(* IEC 61131-3 sources: std_i2980_v2.06_cp053/Source/IMM/ieccontrol/OperationMode1 (part 2) *)

(* ---- ABOperationMode.pu ---- *)
IMPORT_OVER_LISTFILE
 GET_ALARM_NAME
, SET_ALARM
, SET_EVENT
, tnOperationMode
, tsLockOperationModeAuto
, tsTraceLevel
, tnDataState
, ALARM_EVENT
, ABOpModeControl
, tevPanelButtonRegisterData
, tevPanelButtonRegister
, FBDebugTrace
, tsDeviceId
, ALARM_EVENT_DATA

END_IMPORT

ALGORITHM_BLOCK ABOperationMode #DUMMY_EDIT_BLOCK

SYSTEM_VAR
 di_ButtonSetup : BOOL;
 di_ButtonManual : BOOL;
 di_ButtonHalfAuto : BOOL;
 di_ButtonFullAuto : BOOL;
 sv_bButtonSetup : BOOL;
 sv_bButtonManual : BOOL;
 sv_bButtonHalfAuto : BOOL;
 sv_bButtonFullAuto : BOOL;
 sv_bLedManual_ledAttr : BYTE (* Panel LED *);
 sv_bLedSetup_ledAttr : BYTE (* Panel LED *);
 sv_bLedHalfAutomatic_ledAttr : BYTE (* Panel LED *);
 sv_bLedFullAutomatic_ledAttr : BYTE (* Panel LED *);
 sv_DemandedOperationMode : tnOperationMode;
 sv_OperationMode : tnOperationMode;
 sv_bLedSetup : BOOL;
 sv_bLedManual : BOOL;
 sv_bLedHalfAutomatic : BOOL;
 sv_bLedFullAutomatic : BOOL;
 sv_bInitStart : BOOL;
 sv_bAllowFullAutoMode : BOOL;
 sv_bOverrideCoreSafety : BOOL (* overrides safety settings for core movements in setup mode *);
 sv_bOverrideEjectorSafety : BOOL (* overrides safety settings for ejector movements in setup mode *);
 sv_LockOperationModeAuto : tsLockOperationModeAuto;
 sv_TraceLevel : tsTraceLevel;
 sv_DataState : tnDataState (* State of machine / mold data read *);
 sv_DeviceId : tsDeviceId;
 sv_bHMILedManual_ledAttr : BYTE (* Panel LED *);
 sv_bHMILedSetup_ledAttr : BYTE (* Panel LED *);
 sv_bHMILedHalfAutomatic_ledAttr : BYTE (* Panel LED *);
 sv_bHMILedFullAutomatic_ledAttr : BYTE (* Panel LED *);
 sv_bHMILedSetup : BOOL;
 sv_bHMILedManual : BOOL;
 sv_bHMILedHalfAutomatic : BOOL;
 sv_bHMILedFullAutomatic : BOOL;
END_VAR

SYSTEM_OBJECT
 PU_Task_7 : TASK;
 EV_Task_3 : TASK;
 erFullAutoNotAllowed : ALARM;
 erAutoNotAllowed : ALARM;
 erSetupModeRequired : ALARM;
 evAlarmAutoHalf : ALARM_EVENT;
 evAlarmAutoManual : ALARM_EVENT;
 evPanelButtonRegister : tevPanelButtonRegister;
END_OBJECT

VAR
 mbDIButtonManualLinked : BOOL;
 mbDIButtonSetupLinked : BOOL;
 mbDIButtonHalfAutoLinked : BOOL;
 mbDIButtonFullAutoLinked : BOOL;
 mbLedSetupLinked : BOOL;
 mbLedManualLinked : BOOL;
 mbLedHalfAutomaticLinked : BOOL;
 mbLedFullAutomaticLinked : BOOL;
 mbLedSetupAttrLinked : BOOL;
 mbLedManualAttrLinked : BOOL;
 mbLedHalfAutomaticAttrLinked : BOOL;
 mbLedFullAutomaticAttrLinked : BOOL;
 abOpModeControl : ABOpModeControl;
 evPanelButtonRegisterData : tevPanelButtonRegisterData;
 fbDebugTrace : FBDebugTrace;
END_VAR

VAR CONSTANT
 cButtonManual : DINT := 1;
 cButtonSetup : DINT := 2;
 cButtonHalfAuto : DINT := 3;
 cButtonFullAuto : DINT := 4;
END_VAR

POSTUPDATE_ALGORITHM pRegisterButtons ON PU_Task_7 WITH sv_bInitStart

#BEGIN_EDIT_BLOCK
(**************************************** WARNING ********************************************
 *** The KEBA Kemro K2 System including software is not intended for safety control tasks! ***
 ***                       For further information see Comment tab!                        ***
 *********************************************************************************************)

mbDIButtonManualLinked := IS_LINKED(di_ButtonManual);
mbDIButtonSetupLinked := IS_LINKED(di_ButtonSetup);
mbDIButtonHalfAutoLinked  := IS_LINKED(di_ButtonHalfAuto);
mbDIButtonFullAutoLinked := IS_LINKED(di_ButtonFullAuto);

// register manual button
evPanelButtonRegisterData.Button.nPanelButtonType := nPanelButtonAction;
evPanelButtonRegisterData.Button.iCompId := sv_DeviceId.CompId;
evPanelButtonRegisterData.Button.iIndexId := sv_DeviceId.IndexId;
evPanelButtonRegisterData.Button.iButtonId := cButtonManual;
evPanelButtonRegisterData.Button.pbActionVar1 := @sv_bButtonManual;
evPanelButtonRegisterData.Button.Optional.pbLedVar := @sv_bHMILedManual;
evPanelButtonRegisterData.Button.Optional.piLedVarAttr := @sv_bHMILedManual_ledAttr;
SET_EVENT(evPanelButtonRegister, evPanelButtonRegisterData);

// register setup button
evPanelButtonRegisterData.Button.nPanelButtonType := nPanelButtonAction;
evPanelButtonRegisterData.Button.iCompId := sv_DeviceId.CompId;
evPanelButtonRegisterData.Button.iIndexId := sv_DeviceId.IndexId;
evPanelButtonRegisterData.Button.iButtonId := cButtonSetup;
evPanelButtonRegisterData.Button.pbActionVar1 := @sv_bButtonSetup;
evPanelButtonRegisterData.Button.Optional.pbLedVar := @sv_bHMILedSetup;
evPanelButtonRegisterData.Button.Optional.piLedVarAttr := @sv_bHMILedSetup_ledAttr;
SET_EVENT(evPanelButtonRegister, evPanelButtonRegisterData);

// register half-auto button
evPanelButtonRegisterData.Button.nPanelButtonType := nPanelButtonAction;
evPanelButtonRegisterData.Button.iCompId := sv_DeviceId.CompId;
evPanelButtonRegisterData.Button.iIndexId := sv_DeviceId.IndexId;
evPanelButtonRegisterData.Button.iButtonId := cButtonHalfAuto;
evPanelButtonRegisterData.Button.pbActionVar1 := @sv_bButtonHalfAuto;
evPanelButtonRegisterData.Button.Optional.pbLedVar := @sv_bHMILedHalfAutomatic;
evPanelButtonRegisterData.Button.Optional.piLedVarAttr := @sv_bHMILedHalfAutomatic_ledAttr;
SET_EVENT(evPanelButtonRegister, evPanelButtonRegisterData);

// register full-auto button
evPanelButtonRegisterData.Button.nPanelButtonType := nPanelButtonAction;
evPanelButtonRegisterData.Button.iCompId := sv_DeviceId.CompId;
evPanelButtonRegisterData.Button.iIndexId := sv_DeviceId.IndexId;
evPanelButtonRegisterData.Button.iButtonId := cButtonFullAuto;
evPanelButtonRegisterData.Button.pbActionVar1 := @sv_bButtonFullAuto;
evPanelButtonRegisterData.Button.Optional.pbLedVar := @sv_bHMILedFullAutomatic;
evPanelButtonRegisterData.Button.Optional.piLedVarAttr := @sv_bHMILedFullAutomatic_ledAttr;
SET_EVENT(evPanelButtonRegister, evPanelButtonRegisterData);

;#END_EDIT_BLOCK END_ALGORITHM

POSTUPDATE_ALGORITHM pOpModeButton ON PU_Task_7 WITH di_ButtonSetup,di_ButtonManual,di_ButtonHalfAuto,di_ButtonFullAuto,sv_bButtonSetup,sv_bButtonManual,sv_bButtonHalfAuto,sv_bButtonFullAuto

VAR
 bButtonSetup : BOOL;
 bButtonManual : BOOL;
 bButtonHalfAuto : BOOL;
 bButtonFullAuto : BOOL;
END_VAR
#BEGIN_EDIT_BLOCK
(**************************************** WARNING ********************************************
 *** The KEBA Kemro K2 System including software is not intended for safety control tasks! ***
 ***                       For further information see Comment tab!                        ***
 *********************************************************************************************)

//set demanded operation mode according the pressed button

bButtonManual := sv_bButtonManual;
bButtonSetup := sv_bButtonSetup;
bButtonHalfAuto := sv_bButtonHalfAuto;
bButtonFullAuto := sv_bButtonFullAuto;

IF mbDIButtonManualLinked THEN
    bButtonManual := bButtonManual OR di_ButtonManual;
END_IF;

IF mbDIButtonSetupLinked THEN
    bButtonSetup := bButtonSetup OR di_ButtonSetup;
END_IF;

IF mbDIButtonHalfAutoLinked THEN
    bButtonHalfAuto := bButtonHalfAuto OR di_ButtonHalfAuto;
END_IF;

IF mbDIButtonFullAutoLinked THEN
    bButtonFullAuto := bButtonFullAuto OR di_ButtonFullAuto;
END_IF;

IF bButtonSetup THEN
    sv_DemandedOperationMode := nSetup;
ELSIF bButtonManual THEN
    sv_DemandedOperationMode := nManual;
ELSIF bButtonHalfAuto THEN
    sv_DemandedOperationMode := nHalfAutomatic;
ELSIF bButtonFullAuto THEN
    sv_DemandedOperationMode := nFullAutomatic;
END_IF;

;#END_EDIT_BLOCK END_ALGORITHM

POSTUPDATE_ALGORITHM pNewDemandedMode ON PU_Task_7 WITH sv_DemandedOperationMode

VAR_TEMP
 sDemandedOperationMode : STRING(255);
END_VAR
#BEGIN_EDIT_BLOCK
(**************************************** WARNING ********************************************
 *** The KEBA Kemro K2 System including software is not intended for safety control tasks! ***
 ***                       For further information see Comment tab!                        ***
 *********************************************************************************************)

IF sv_DemandedOperationMode = sv_OperationMode THEN
    //don´t execute if operation mode is equal demanded operation mode
    RETURN;
END_IF;

IF sv_TraceLevel.bODCInterpreter THEN
   //trace demanded opmode switch
   IF sv_DemandedOperationMode = nSetup THEN
      sDemandedOperationMode := 'Setup';
   ELSIF sv_DemandedOperationMode = nManual THEN
      sDemandedOperationMode := 'Manual';
   ELSIF sv_DemandedOperationMode = nHalfAutomatic THEN
      sDemandedOperationMode := 'HalfAutomatic';
   ELSIF sv_DemandedOperationMode = nFullAutomatic THEN
      sDemandedOperationMode := 'FullAutomatic';
   ELSE
      sDemandedOperationMode := '???';
   END_IF;
   fbDebugTrace(CONCAT('sv_DemandedOperationMode changed to ', sDemandedOperationMode));
END_IF;

IF sv_DemandedOperationMode = nFullAutomatic AND NOT sv_bAllowFullAutoMode THEN
    //change to full auto mode not allowed
    SET_ALARM (Name := erFullAutoNotAllowed);
    sv_DemandedOperationMode := sv_OperationMode;
    IF sv_TraceLevel.bODCInterpreter THEN
        fbDebugTrace('operation mode switch denied by sv_bAllowFullAutoMode');
    END_IF;
    RETURN;
END_IF;

// if demanded mode (half)automatic check if data loading is active
IF (sv_DemandedOperationMode > nManual) THEN
    IF ((sv_DataState = nReadMoldData)
        OR (sv_DataState = nReadMachineData)
        OR (sv_DataState = nReadSequenceData)
        OR (sv_DataState = nReadMaterialData)) THEN
        SET_ALARM(erAutoNotAllowed);
        sv_DemandedOperationMode := sv_OperationMode;
        IF sv_TraceLevel.bODCInterpreter THEN
            fbDebugTrace('operation mode switch denied by data loading');
        END_IF;
        RETURN;
    END_IF;
    IF (sv_LockOperationModeAuto.iLockCounter > 0) THEN
        SET_ALARM(erAutoNotAllowed);
        sv_DemandedOperationMode := sv_OperationMode;
        IF sv_TraceLevel.bODCInterpreter THEN
            fbDebugTrace('operation mode switch denied by data sv_LockOperationModeAuto');
        END_IF;
        RETURN;
    END_IF;
END_IF;

//check if demanded operation mode is allowed
abOpModeControl.aCheck(nDemandedMode := sv_DemandedOperationMode,
                       nActualMode := sv_OperationMode);

IF abOpModeControl.aCheck.bChangeAllowed THEN
    //change allowed
    sv_OperationMode := sv_DemandedOperationMode;
ELSE
    //change not allowed
    sv_DemandedOperationMode := sv_OperationMode;
    IF sv_TraceLevel.bODCInterpreter THEN
        fbDebugTrace('operation mode switch denied by abOpModeControl.aCheck()');
    END_IF;
END_IF;

;#END_EDIT_BLOCK END_ALGORITHM

POSTUPDATE_ALGORITHM pLedControl ON PU_Task_7 WITH sv_OperationMode, sv_bInitStart

VAR
 bInitDone : BOOL;
END_VAR
#BEGIN_EDIT_BLOCK
(**************************************** WARNING ********************************************
 *** The KEBA Kemro K2 System including software is not intended for safety control tasks! ***
 ***                       For further information see Comment tab!                        ***
 *********************************************************************************************)

IF NOT bInitDone THEN
   //set HMI button led system variables
   sv_bHMILedSetup_ledAttr := 16#1;
   sv_bHMILedManual_ledAttr := 16#1;
   sv_bHMILedHalfAutomatic_ledAttr := 16#1;
   sv_bHMILedFullAutomatic_ledAttr := 16#1;

   mbLedSetupLinked := IS_LINKED(sv_bLedSetup);
   mbLedManualLinked := IS_LINKED(sv_bLedManual);
   mbLedHalfAutomaticLinked := IS_LINKED(sv_bLedHalfAutomatic);
   mbLedFullAutomaticLinked := IS_LINKED(sv_bLedFullAutomatic);

   //set led attributes
   IF IS_LINKED(sv_bLedSetup_ledAttr) THEN
      sv_bLedSetup_ledAttr := sv_bHMILedSetup_ledAttr;
      mbLedSetupAttrLinked := TRUE;
   END_IF;

   IF IS_LINKED(sv_bLedManual_ledAttr) THEN
      sv_bLedManual_ledAttr := sv_bHMILedManual_ledAttr;
      mbLedManualAttrLinked := TRUE;
   END_IF;

   IF IS_LINKED(sv_bLedHalfAutomatic_ledAttr) THEN
      sv_bLedHalfAutomatic_ledAttr := sv_bHMILedHalfAutomatic_ledAttr;
      mbLedHalfAutomaticAttrLinked := TRUE;
   END_IF;

   IF IS_LINKED(sv_bLedFullAutomatic_ledAttr) THEN
      sv_bLedFullAutomatic_ledAttr := sv_bHMILedFullAutomatic_ledAttr;
      mbLedFullAutomaticAttrLinked := TRUE;
   END_IF;

   bInitDone := TRUE;
END_IF;

IF (sv_OperationMode = nManual) THEN
   sv_bHMILedManual := TRUE;
   sv_bHMILedSetup := FALSE;
   sv_bHMILedHalfAutomatic := FALSE;
   sv_bHMILedFullAutomatic := FALSE;

ELSIF (sv_OperationMode = nSetup) THEN
   sv_bHMILedManual := FALSE;
   sv_bHMILedSetup := TRUE;
   sv_bHMILedHalfAutomatic := FALSE;
   sv_bHMILedFullAutomatic := FALSE;

ELSIF (sv_OperationMode = nHalfAutomatic) THEN
   sv_bHMILedManual := FALSE;
   sv_bHMILedSetup := FALSE;
   sv_bHMILedHalfAutomatic := TRUE;
   sv_bHMILedFullAutomatic := FALSE;

ELSIF (sv_OperationMode = nFullAutomatic) THEN
   sv_bHMILedManual := FALSE;
   sv_bHMILedSetup := FALSE;
   sv_bHMILedHalfAutomatic := FALSE;
   sv_bHMILedFullAutomatic := TRUE;

END_IF;

// copy the led states to the hw-leds
IF mbLedSetupLinked THEN
   sv_bLedSetup := sv_bHMILedSetup;
END_IF;

IF mbLedManualLinked THEN
   sv_bLedManual := sv_bHMILedManual;
END_IF;

IF mbLedHalfAutomaticLinked THEN
   sv_bLedHalfAutomatic := sv_bHMILedHalfAutomatic;
END_IF;

IF mbLedFullAutomaticLinked THEN
   sv_bLedFullAutomatic := sv_bHMILedFullAutomatic;
END_IF;

;#END_EDIT_BLOCK END_ALGORITHM

EVENT_ALGORITHM evaAlarmAutoManual ON EV_Task_3 WITH evAlarmAutoManual

VAR_INPUT
 evAlarmAutoManualData : ALARM_EVENT_DATA;
END_VAR
#BEGIN_EDIT_BLOCK
(**************************************** WARNING ********************************************
 *** The KEBA Kemro K2 System including software is not intended for safety control tasks! ***
 ***                       For further information see Comment tab!                        ***
 *********************************************************************************************)

//do not change mode if operation mode is already manual or setup
IF sv_OperationMode >= nHalfAutomatic THEN
   IF sv_TraceLevel.bODCInterpreter THEN
      fbDebugTrace(CONCAT('switching opmode to manual because of evAlarmAutoManual (',
                          GET_ALARM_NAME(evAlarmAutoManualData.NAME), ')'));
   END_IF;
   sv_DemandedOperationMode := nManual;
END_IF;

;#END_EDIT_BLOCK END_ALGORITHM

EVENT_ALGORITHM evaAlarmAutoHalf ON EV_Task_3 WITH evAlarmAutoHalf

VAR_INPUT
 evAlarmAutoManualData : ALARM_EVENT_DATA;
END_VAR
#BEGIN_EDIT_BLOCK
(**************************************** WARNING ********************************************
 *** The KEBA Kemro K2 System including software is not intended for safety control tasks! ***
 ***                       For further information see Comment tab!                        ***
 *********************************************************************************************)

//do not change mode if operation mode is already not full auto
IF sv_OperationMode = nFullAutomatic THEN
   IF sv_TraceLevel.bODCInterpreter THEN
      fbDebugTrace(CONCAT('switching opmode to half auto because of evAlarmAutoHalf (',
                          GET_ALARM_NAME(evAlarmAutoManualData.NAME), ')'));
   END_IF;
   sv_DemandedOperationMode := nHalfAutomatic;
END_IF;

;#END_EDIT_BLOCK END_ALGORITHM

POSTUPDATE_ALGORITHM pOverrideSafety ON PU_Task_7 WITH sv_bOverrideCoreSafety,sv_bOverrideEjectorSafety

#BEGIN_EDIT_BLOCK
(**************************************** WARNING ********************************************
 *** The KEBA Kemro K2 System including software is not intended for safety control tasks! ***
 ***                       For further information see Comment tab!                        ***
 *********************************************************************************************)

IF (sv_OperationMode <> nSetup) THEN
   IF sv_bOverrideCoreSafety THEN
      //reset override core safety flag if mode is not setup mode
      //and set alarm
      sv_bOverrideCoreSafety := FALSE;
      SET_ALARM(erSetupModeRequired);
   END_IF;

   IF sv_bOverrideEjectorSafety THEN
      //reset override ejector safety flag if mode is not setup mode
      //and set alarm
      sv_bOverrideEjectorSafety := FALSE;
      SET_ALARM(erSetupModeRequired);
   END_IF;
END_IF;

;#END_EDIT_BLOCK END_ALGORITHM

POSTUPDATE_ALGORITHM pOperationMode ON PU_Task_7 WITH sv_OperationMode

#BEGIN_EDIT_BLOCK
(**************************************** WARNING ********************************************
 *** The KEBA Kemro K2 System including software is not intended for safety control tasks! ***
 ***                       For further information see Comment tab!                        ***
 *********************************************************************************************)

IF sv_OperationMode <> nSetup THEN
   //reset "override safety" flags if setup mode is left
   sv_bOverrideCoreSafety := FALSE;
   sv_bOverrideEjectorSafety := FALSE;
END_IF;

;#END_EDIT_BLOCK END_ALGORITHM

END_ALGORITHM_BLOCK

#END_OF_IEC_PART

@Puma @IecEditor 6 97 @Pou 25
@@@BEG_Comment@@@

@@@END_Comment@@@

@BEG_Contents

@BEG_Func
@RT(17)FuncTreeContainer
3
@Var @RT(14)GET_ALARM_NAME @RT(0) @T @T @DERIVED 0 @F @RT(22)KEBA_STANDARD_FUNCTION @F
@T
@BEG_Attrib
0 @RT(0) @RT(0)
@END_Attrib
1 1 @F @F @F @F

@Var @RT(9)SET_ALARM @RT(0) @T @T @DERIVED 0 @F @RT(23)KEBA_STANDARD_PROCEDURE @F
@T
@BEG_Attrib
0 @RT(0) @RT(0)
@END_Attrib
1 1 @F @F @F @F

@Var @RT(9)SET_EVENT @RT(0) @T @T @DERIVED 0 @F @RT(23)KEBA_STANDARD_PROCEDURE @F
@T
@BEG_Attrib
0 @RT(0) @RT(0)
@END_Attrib
1 1 @F @F @F @F

@END_Func

@BEG_Const
@RT(18)ConstTreeContainer
0
@END_Const

@BEG_Export

@BEG_Kind
@ALGORITHM_BLOCK @RT(15)ABOperationMode @STRUCTURED_TEXT
@RT(0) @RT(0) @RT(0)
@END_Kind

@BEG_Dcl
@RT(16)DclTreeContainer
61
@Var @RT(14)di_ButtonSetup @RT(0) @T @F @DT @RT(4)BOOL @RT(0) @T @T @BASIC 0 @F
@F @F
@T
@BEG_Attrib
3 @RT(0) @RT(0) @RT(0)
@END_Attrib
1 8 @F @F @F @F

@Var @RT(15)di_ButtonManual @RT(0) @T @F @DT @RT(4)BOOL @RT(0) @T @T @BASIC 0 @F
@F @F
@T
@BEG_Attrib
3 @RT(0) @RT(0) @RT(0)
@END_Attrib
1 8 @F @F @F @F

@Var @RT(17)di_ButtonHalfAuto @RT(0) @T @F @DT @RT(4)BOOL @RT(0) @T @T @BASIC 0 @F
@F @F
@T
@BEG_Attrib
3 @RT(0) @RT(0) @RT(0)
@END_Attrib
1 8 @F @F @F @F

@Var @RT(17)di_ButtonFullAuto @RT(0) @T @F @DT @RT(4)BOOL @RT(0) @T @T @BASIC 0 @F
@F @F
@T
@BEG_Attrib
3 @RT(0) @RT(0) @RT(0)
@END_Attrib
1 8 @F @F @F @F

@Var @RT(22)mbDIButtonManualLinked @RT(0) @T @F @DT @RT(4)BOOL @RT(0) @T @T @BASIC 0 @F
@F @F
@T
@BEG_Attrib
3 @RT(0) @RT(0) @RT(0)
@END_Attrib
1 0 @F @F @F @F

@Var @RT(21)mbDIButtonSetupLinked @RT(0) @T @F @DT @RT(4)BOOL @RT(0) @T @T @BASIC 0 @F
@F @F
@T
@BEG_Attrib
3 @RT(0) @RT(0) @RT(0)
@END_Attrib
1 0 @F @F @F @F

@Var @RT(24)mbDIButtonHalfAutoLinked @RT(0) @T @F @DT @RT(4)BOOL @RT(0) @T @T @BASIC 0 @F
@F @F
@T
@BEG_Attrib
3 @RT(0) @RT(0) @RT(0)
@END_Attrib
1 0 @F @F @F @F

@Var @RT(24)mbDIButtonFullAutoLinked @RT(0) @T @F @DT @RT(4)BOOL @RT(0) @T @T @BASIC 0 @F
@F @F
@T
@BEG_Attrib
3 @RT(0) @RT(0) @RT(0)
@END_Attrib
1 0 @F @F @F @F

@Var @RT(16)mbLedSetupLinked @RT(0) @T @F @DT @RT(4)BOOL @RT(0) @T @T @BASIC 0 @F
@F @F
@T
@BEG_Attrib
3 @RT(0) @RT(0) @RT(0)
@END_Attrib
1 0 @F @F @F @F

@Var @RT(17)mbLedManualLinked @RT(0) @T @F @DT @RT(4)BOOL @RT(0) @T @T @BASIC 0 @F
@F @F
@T
@BEG_Attrib
3 @RT(0) @RT(0) @RT(0)
@END_Attrib
1 0 @F @F @F @F

@Var @RT(24)mbLedHalfAutomaticLinked @RT(0) @T @F @DT @RT(4)BOOL @RT(0) @T @T @BASIC 0 @F
@F @F
@T
@BEG_Attrib
3 @RT(0) @RT(0) @RT(0)
@END_Attrib
1 0 @F @F @F @F

@Var @RT(24)mbLedFullAutomaticLinked @RT(0) @T @F @DT @RT(4)BOOL @RT(0) @T @T @BASIC 0 @F
@F @F
@T
@BEG_Attrib
3 @RT(0) @RT(0) @RT(0)
@END_Attrib
1 0 @F @F @F @F

@Var @RT(20)mbLedSetupAttrLinked @RT(0) @T @F @DT @RT(4)BOOL @RT(0) @T @T @BASIC 0 @F
@F @F
@T
@BEG_Attrib
3 @RT(0) @RT(0) @RT(0)
@END_Attrib
1 0 @F @F @F @F

@Var @RT(21)mbLedManualAttrLinked @RT(0) @T @F @DT @RT(4)BOOL @RT(0) @T @T @BASIC 0 @F
@F @F
@T
@BEG_Attrib
3 @RT(0) @RT(0) @RT(0)
@END_Attrib
1 0 @F @F @F @F

@Var @RT(28)mbLedHalfAutomaticAttrLinked @RT(0) @T @F @DT @RT(4)BOOL @RT(0) @T @T @BASIC 0 @F
@F @F
@T
@BEG_Attrib
3 @RT(0) @RT(0) @RT(0)
@END_Attrib
1 0 @F @F @F @F

@Var @RT(28)mbLedFullAutomaticAttrLinked @RT(0) @T @F @DT @RT(4)BOOL @RT(0) @T @T @BASIC 0 @F
@F @F
@T
@BEG_Attrib
3 @RT(0) @RT(0) @RT(0)
@END_Attrib
1 0 @F @F @F @F

@Var @RT(15)sv_bButtonSetup @RT(0) @T @F @DT @RT(4)BOOL @RT(0) @T @T @BASIC 0 @F
@F @F
@T
@BEG_Attrib
3 @RT(0) @RT(0) @RT(0)
@END_Attrib
1 8 @F @F @F @F

@Var @RT(16)sv_bButtonManual @RT(0) @T @F @DT @RT(4)BOOL @RT(0) @T @T @BASIC 0 @F
@F @F
@T
@BEG_Attrib
3 @RT(0) @RT(0) @RT(0)
@END_Attrib
1 8 @F @F @F @F

@Var @RT(18)sv_bButtonHalfAuto @RT(0) @T @F @DT @RT(4)BOOL @RT(0) @T @T @BASIC 0 @F
@F @F
@T
@BEG_Attrib
3 @RT(0) @RT(0) @RT(0)
@END_Attrib
1 8 @F @F @F @F

@Var @RT(18)sv_bButtonFullAuto @RT(0) @T @F @DT @RT(4)BOOL @RT(0) @T @T @BASIC 0 @F
@F @F
@T
@BEG_Attrib
3 @RT(0) @RT(0) @RT(0)
@END_Attrib
1 8 @F @F @F @F

@Var @RT(21)sv_bLedManual_ledAttr @RT(0) @T @F @DT @RT(4)BYTE @RT(0) @T @T @BASIC 0 @F
@F @F
@T
@BEG_Attrib
3 @RT(0) @RT(9)Panel LED @RT(0)
@END_Attrib
1 8 @F @F @F @F

@Var @RT(20)sv_bLedSetup_ledAttr @RT(0) @T @F @DT @RT(4)BYTE @RT(0) @T @T @BASIC 0 @F
@F @F
@T
@BEG_Attrib
3 @RT(0) @RT(9)Panel LED @RT(0)
@END_Attrib
1 8 @F @F @F @F

@Var @RT(28)sv_bLedHalfAutomatic_ledAttr @RT(0) @T @F @DT @RT(4)BYTE @RT(0) @T @T @BASIC 0 @F
@F @F
@T
@BEG_Attrib
3 @RT(0) @RT(9)Panel LED @RT(0)
@END_Attrib
1 8 @F @F @F @F

@Var @RT(28)sv_bLedFullAutomatic_ledAttr @RT(0) @T @F @DT @RT(4)BYTE @RT(0) @T @T @BASIC 0 @F
@F @F
@T
@BEG_Attrib
3 @RT(0) @RT(9)Panel LED @RT(0)
@END_Attrib
1 8 @F @F @F @F

@Var @RT(24)sv_DemandedOperationMode @RT(0) @T @T @DERIVED 0 @T @T @DT @RT(15)tnOperationMode @RT(0) @T @T @UNKNOWN 0 @F
@F @F
@T
@BEG_Attrib
3 @RT(0) @RT(0) @RT(0)
@END_Attrib
1 8 @F @F @F @F

@Var @RT(16)sv_OperationMode @RT(0) @T @T @DERIVED 0 @T @T @DT @RT(15)tnOperationMode @RT(0) @T @T @UNKNOWN 0 @F
@F @F
@T
@BEG_Attrib
3 @RT(0) @RT(0) @RT(0)
@END_Attrib
1 8 @F @F @F @F

@Var @RT(12)sv_bLedSetup @RT(0) @T @F @DT @RT(4)BOOL @RT(0) @T @T @BASIC 0 @F
@F @F
@T
@BEG_Attrib
3 @RT(0) @RT(0) @RT(0)
@END_Attrib
1 8 @F @F @F @F

@Var @RT(13)sv_bLedManual @RT(0) @T @F @DT @RT(4)BOOL @RT(0) @T @T @BASIC 0 @F
@F @F
@T
@BEG_Attrib
3 @RT(0) @RT(0) @RT(0)
@END_Attrib
1 8 @F @F @F @F

@Var @RT(20)sv_bLedHalfAutomatic @RT(0) @T @F @DT @RT(4)BOOL @RT(0) @T @T @BASIC 0 @F
@F @F
@T
@BEG_Attrib
3 @RT(0) @RT(0) @RT(0)
@END_Attrib
1 8 @F @F @F @F

@Var @RT(20)sv_bLedFullAutomatic @RT(0) @T @F @DT @RT(4)BOOL @RT(0) @T @T @BASIC 0 @F
@F @F
@T
@BEG_Attrib
3 @RT(0) @RT(0) @RT(0)
@END_Attrib
1 8 @F @F @F @F

@Var @RT(13)sv_bInitStart @RT(0) @T @F @DT @RT(4)BOOL @RT(0) @T @T @BASIC 0 @F
@F @F
@T
@BEG_Attrib
3 @RT(0) @RT(0) @RT(0)
@END_Attrib
1 8 @F @F @F @F

@Var @RT(21)sv_bAllowFullAutoMode @RT(0) @T @F @DT @RT(4)BOOL @RT(0) @T @T @BASIC 0 @F
@F @F
@T
@BEG_Attrib
3 @RT(0) @RT(0) @RT(0)
@END_Attrib
1 8 @F @F @F @F

@Var @RT(22)sv_bOverrideCoreSafety @RT(0) @T @F @DT @RT(4)BOOL @RT(0) @T @T @BASIC 0 @F
@F @F
@T
@BEG_Attrib
3 @RT(0) @RT(58)overrides safety settings for core movements in setup mode @RT(0)
@END_Attrib
1 8 @F @F @F @F

@Var @RT(25)sv_bOverrideEjectorSafety @RT(0) @T @F @DT @RT(4)BOOL @RT(0) @T @T @BASIC 0 @F
@F @F
@T
@BEG_Attrib
3 @RT(0) @RT(61)overrides safety settings for ejector movements in setup mode @RT(0)
@END_Attrib
1 8 @F @F @F @F

@Var @RT(24)sv_LockOperationModeAuto @RT(0) @T @T @DERIVED 0 @T @T @DT @RT(23)tsLockOperationModeAuto @RT(0) @T @T @UNKNOWN 0 @F
@F @F
@T
@BEG_Attrib
3 @RT(0) @RT(0) @RT(0)
@END_Attrib
1 8 @F @F @F @F

@Var @RT(13)sv_TraceLevel @RT(0) @T @T @RENAMED 0 @T @T @DT @RT(12)tsTraceLevel @RT(0) @T @T @UNKNOWN 0 @F
@F @F
@T
@BEG_Attrib
3 @RT(0) @RT(0) @RT(0)
@END_Attrib
1 8 @F @F @F @F

@Var @RT(9)PU_Task_7 @RT(0) @T @T @RENAMED 0 @T @T @DT @RT(4)TASK @RT(0) @T @T @BASIC 0 @F
@F @F
@T
@BEG_Attrib
3 @RT(0) @RT(0) @RT(0)
@END_Attrib
1 7 @F @F @F @F

@Var @RT(9)EV_Task_3 @RT(0) @T @T @RENAMED 0 @T @T @DT @RT(4)TASK @RT(0) @T @T @BASIC 0 @F
@F @F
@T
@BEG_Attrib
3 @RT(0) @RT(0) @RT(0)
@END_Attrib
1 7 @F @F @F @F

@Var @RT(20)erFullAutoNotAllowed @RT(0) @T @F @DT @RT(5)ALARM @RT(0) @T @T @BASIC 0 @F
@F @F
@T
@BEG_Attrib
3 @RT(0) @RT(0) @RT(0)
@END_Attrib
1 7 @F @F @F @F

@Var @RT(12)sv_DataState @RT(0) @T @T @DERIVED 0 @T @T @DT @RT(11)tnDataState @RT(0) @T @T @UNKNOWN 0 @F
@F @F
@T
@BEG_Attrib
3 @RT(0) @RT(33)State of machine / mold data read @RT(0)
@END_Attrib
1 8 @F @F @F @F

@Var @RT(16)erAutoNotAllowed @RT(0) @T @F @DT @RT(5)ALARM @RT(0) @T @T @BASIC 0 @F
@F @F
@T
@BEG_Attrib
3 @RT(0) @RT(0) @RT(0)
@END_Attrib
1 7 @F @F @F @F

@Var @RT(19)erSetupModeRequired @RT(0) @T @T @RENAMED 0 @T @T @DT @RT(5)ALARM @RT(0) @T @T @BASIC 0 @F
@F @F
@T
@BEG_Attrib
3 @RT(0) @RT(0) @RT(0)
@END_Attrib
1 7 @F @F @F @F

@Var @RT(15)evAlarmAutoHalf @RT(0) @T @T @DERIVED 0 @T @T @DT @RT(11)ALARM_EVENT @RT(0) @T @T @UNKNOWN 0 @F
@F @F
@T
@BEG_Attrib
3 @RT(0) @RT(0) @RT(0)
@END_Attrib
1 7 @F @F @F @F

@Var @RT(17)evAlarmAutoManual @RT(0) @T @T @RENAMED 0 @T @T @DT @RT(11)ALARM_EVENT @RT(0) @T @T @UNKNOWN 0 @F
@F @F
@T
@BEG_Attrib
3 @RT(0) @RT(0) @RT(0)
@END_Attrib
1 7 @F @F @F @F

@Var @RT(15)abOpModeControl @RT(0) @T @T @DERIVED 0 @T @T @DT @RT(15)ABOpModeControl @RT(0) @T @T @UNKNOWN 0 @F
@F @F
@T
@BEG_Attrib
3 @RT(0) @RT(0) @RT(0)
@END_Attrib
1 0 @F @F @F @F

@Var @RT(25)evPanelButtonRegisterData @RT(0) @T @T @DERIVED 0 @T @T @DT @RT(26)tevPanelButtonRegisterData @RT(0) @T @T @UNKNOWN 0 @F
@F @F
@T
@BEG_Attrib
3 @RT(0) @RT(0) @RT(0)
@END_Attrib
1 0 @F @F @F @F

@Var @RT(21)evPanelButtonRegister @RT(0) @T @T @DERIVED 0 @T @T @DT @RT(22)tevPanelButtonRegister @RT(0) @T @T @UNKNOWN 0 @F
@F @F
@T
@BEG_Attrib
3 @RT(0) @RT(0) @RT(0)
@END_Attrib
1 7 @F @F @F @F

@Var @RT(12)fbDebugTrace @RT(0) @T @T @DERIVED 0 @T @T @DT @RT(12)FBDebugTrace @RT(0) @T @T @UNKNOWN 0 @F
@F @F
@T
@BEG_Attrib
3 @RT(0) @RT(0) @RT(0)
@END_Attrib
1 0 @F @F @F @F

@Var @RT(11)sv_DeviceId @RT(0) @T @T @DERIVED 0 @T @T @DT @RT(10)tsDeviceId @RT(0) @T @T @UNKNOWN 0 @F
@F @F
@T
@BEG_Attrib
3 @RT(0) @RT(0) @RT(0)
@END_Attrib
1 8 @F @F @F @F

@Var @RT(13)cButtonManual @RT(0) @T @F @DT @RT(4)DINT @RT(0) @T @T @BASIC 0 @F
@F @F
@T
@BEG_Attrib
3 @RT(1)1 @RT(0) @RT(0)
@END_Attrib
1 15 @F @F @F @F

@Var @RT(12)cButtonSetup @RT(0) @T @F @DT @RT(4)DINT @RT(0) @T @T @BASIC 0 @F
@F @F
@T
@BEG_Attrib
3 @RT(1)2 @RT(0) @RT(0)
@END_Attrib
1 15 @F @F @F @F

@Var @RT(15)cButtonHalfAuto @RT(0) @T @F @DT @RT(4)DINT @RT(0) @T @T @BASIC 0 @F
@F @F
@T
@BEG_Attrib
3 @RT(1)3 @RT(0) @RT(0)
@END_Attrib
1 15 @F @F @F @F

@Var @RT(15)cButtonFullAuto @RT(0) @T @F @DT @RT(4)DINT @RT(0) @T @T @BASIC 0 @F
@F @F
@T
@BEG_Attrib
3 @RT(1)4 @RT(0) @RT(0)
@END_Attrib
1 15 @F @F @F @F

@Var @RT(24)sv_bHMILedManual_ledAttr @RT(0) @T @F @DT @RT(4)BYTE @RT(0) @T @T @BASIC 0 @F
@F @F
@T
@BEG_Attrib
3 @RT(0) @RT(9)Panel LED @RT(0)
@END_Attrib
1 8 @F @F @F @F

@Var @RT(23)sv_bHMILedSetup_ledAttr @RT(0) @T @F @DT @RT(4)BYTE @RT(0) @T @T @BASIC 0 @F
@F @F
@T
@BEG_Attrib
3 @RT(0) @RT(9)Panel LED @RT(0)
@END_Attrib
1 8 @F @F @F @F

@Var @RT(31)sv_bHMILedHalfAutomatic_ledAttr @RT(0) @T @F @DT @RT(4)BYTE @RT(0) @T @T @BASIC 0 @F
@F @F
@T
@BEG_Attrib
3 @RT(0) @RT(9)Panel LED @RT(0)
@END_Attrib
1 8 @F @F @F @F

@Var @RT(31)sv_bHMILedFullAutomatic_ledAttr @RT(0) @T @F @DT @RT(4)BYTE @RT(0) @T @T @BASIC 0 @F
@F @F
@T
@BEG_Attrib
3 @RT(0) @RT(9)Panel LED @RT(0)
@END_Attrib
1 8 @F @F @F @F

@Var @RT(15)sv_bHMILedSetup @RT(0) @T @F @DT @RT(4)BOOL @RT(0) @T @T @BASIC 0 @F
@F @F
@T
@BEG_Attrib
3 @RT(0) @RT(0) @RT(0)
@END_Attrib
1 8 @F @F @F @F

@Var @RT(16)sv_bHMILedManual @RT(0) @T @F @DT @RT(4)BOOL @RT(0) @T @T @BASIC 0 @F
@F @F
@T
@BEG_Attrib
3 @RT(0) @RT(0) @RT(0)
@END_Attrib
1 8 @F @F @F @F

@Var @RT(23)sv_bHMILedHalfAutomatic @RT(0) @T @F @DT @RT(4)BOOL @RT(0) @T @T @BASIC 0 @F
@F @F
@T
@BEG_Attrib
3 @RT(0) @RT(0) @RT(0)
@END_Attrib
1 8 @F @F @F @F

@Var @RT(23)sv_bHMILedFullAutomatic @RT(0) @T @F @DT @RT(4)BOOL @RT(0) @T @T @BASIC 0 @F
@F @F
@T
@BEG_Attrib
3 @RT(0) @RT(0) @RT(0)
@END_Attrib
1 8 @F @F @F @F

@END_Dcl

@END_Export

@BEG_Body

8

@BEG_Export

@BEG_Algo
@POSTUPDATE_ALGORITHM @RT(16)pRegisterButtons @STRUCTURED_TEXT
@RT(0) @RT(13)sv_bInitStart @RT(9)PU_Task_7 @F @F
@END_Algo

@BEG_Dcl
@RT(16)DclTreeContainer
0
@END_Dcl

@END_Export

@BEG_Export

@BEG_Algo
@POSTUPDATE_ALGORITHM @RT(13)pOpModeButton @STRUCTURED_TEXT
@RT(0) @RT(137)di_ButtonSetup,di_ButtonManual,di_ButtonHalfAuto,di_ButtonFullAuto,sv_bButtonSetup,sv_bButtonManual,sv_bButtonHalfAuto,sv_bButtonFullAuto @RT(9)PU_Task_7 @F @F
@END_Algo

@BEG_Dcl
@RT(16)DclTreeContainer
4
@Var @RT(12)bButtonSetup @RT(0) @T @F @DT @RT(4)BOOL @RT(0) @T @T @BASIC 0 @F
@F @F
@T
@BEG_Attrib
3 @RT(0) @RT(0) @RT(0)
@END_Attrib
1 0 @F @F @F @F

@Var @RT(13)bButtonManual @RT(0) @T @F @DT @RT(4)BOOL @RT(0) @T @T @BASIC 0 @F
@F @F
@T
@BEG_Attrib
3 @RT(0) @RT(0) @RT(0)
@END_Attrib
1 0 @F @F @F @F

@Var @RT(15)bButtonHalfAuto @RT(0) @T @F @DT @RT(4)BOOL @RT(0) @T @T @BASIC 0 @F
@F @F
@T
@BEG_Attrib
3 @RT(0) @RT(0) @RT(0)
@END_Attrib
1 0 @F @F @F @F

@Var @RT(15)bButtonFullAuto @RT(0) @T @F @DT @RT(4)BOOL @RT(0) @T @T @BASIC 0 @F
@F @F
@T
@BEG_Attrib
3 @RT(0) @RT(0) @RT(0)
@END_Attrib
1 0 @F @F @F @F

@END_Dcl

@END_Export

@BEG_Export

@BEG_Algo
@POSTUPDATE_ALGORITHM @RT(16)pNewDemandedMode @STRUCTURED_TEXT
@RT(0) @RT(24)sv_DemandedOperationMode @RT(9)PU_Task_7 @F @F
@END_Algo

@BEG_Dcl
@RT(16)DclTreeContainer
1
@Var @RT(22)sDemandedOperationMode @RT(0) @T @F @DT @RT(11)STRING(255) @RT(0) @T @T @STRING 0 @F @RT(3)255 @F
@F @F
@T
@BEG_Attrib
3 @RT(0) @RT(0) @RT(0)
@END_Attrib
1 4 @F @F @F @F

@END_Dcl

@END_Export

@BEG_Export

@BEG_Algo
@POSTUPDATE_ALGORITHM @RT(11)pLedControl @STRUCTURED_TEXT
@RT(0) @RT(31)sv_OperationMode, sv_bInitStart @RT(9)PU_Task_7 @F @F
@END_Algo

@BEG_Dcl
@RT(16)DclTreeContainer
1
@Var @RT(9)bInitDone @RT(0) @T @F @DT @RT(4)BOOL @RT(0) @T @T @BASIC 0 @F
@F @F
@T
@BEG_Attrib
3 @RT(0) @RT(0) @RT(0)
@END_Attrib
1 0 @F @F @F @F

@END_Dcl

@END_Export

@BEG_Export

@BEG_Algo
@EVENT_ALGORITHM @RT(18)evaAlarmAutoManual @STRUCTURED_TEXT
@RT(0) @RT(17)evAlarmAutoManual @RT(9)EV_Task_3 @F @F
@END_Algo

@BEG_Dcl
@RT(16)DclTreeContainer
1
@Var @RT(21)evAlarmAutoManualData @RT(0) @T @T @DERIVED 0 @T @T @DT @RT(16)ALARM_EVENT_DATA @RT(0) @T @T @UNKNOWN 0 @F
@F @F
@T
@BEG_Attrib
3 @RT(0) @RT(0) @RT(0)
@END_Attrib
1 1 @F @F @F @F

@END_Dcl

@END_Export

@BEG_Export

@BEG_Algo
@EVENT_ALGORITHM @RT(16)evaAlarmAutoHalf @STRUCTURED_TEXT
@RT(0) @RT(15)evAlarmAutoHalf @RT(9)EV_Task_3 @F @F
@END_Algo

@BEG_Dcl
@RT(16)DclTreeContainer
1
@Var @RT(21)evAlarmAutoManualData @RT(0) @T @T @DERIVED 0 @T @T @DT @RT(16)ALARM_EVENT_DATA @RT(0) @T @T @UNKNOWN 0 @F
@F @F
@T
@BEG_Attrib
3 @RT(0) @RT(0) @RT(0)
@END_Attrib
1 1 @F @F @F @F

@END_Dcl

@END_Export

@BEG_Export

@BEG_Algo
@POSTUPDATE_ALGORITHM @RT(15)pOverrideSafety @STRUCTURED_TEXT
@RT(0) @RT(48)sv_bOverrideCoreSafety,sv_bOverrideEjectorSafety @RT(9)PU_Task_7 @F @F
@END_Algo

@BEG_Dcl
@RT(16)DclTreeContainer
0
@END_Dcl

@END_Export

@BEG_Export

@BEG_Algo
@POSTUPDATE_ALGORITHM @RT(14)pOperationMode @STRUCTURED_TEXT
@RT(0) @RT(16)sv_OperationMode @RT(9)PU_Task_7 @F @F
@END_Algo

@BEG_Dcl
@RT(16)DclTreeContainer
0
@END_Dcl

@END_Export

@BEG_Body
@TL(54)
(**************************************** WARNING ********************************************
 *** The KEBA Kemro K2 System including software is not intended for safety control tasks! ***
 ***                       For further information see Comment tab!                        ***
 *********************************************************************************************)

mbDIButtonManualLinked := IS_LINKED(di_ButtonManual);
mbDIButtonSetupLinked := IS_LINKED(di_ButtonSetup);
mbDIButtonHalfAutoLinked  := IS_LINKED(di_ButtonHalfAuto);
mbDIButtonFullAutoLinked := IS_LINKED(di_ButtonFullAuto);

// register manual button
evPanelButtonRegisterData.Button.nPanelButtonType := nPanelButtonAction;
evPanelButtonRegisterData.Button.iCompId := sv_DeviceId.CompId;
evPanelButtonRegisterData.Button.iIndexId := sv_DeviceId.IndexId;
evPanelButtonRegisterData.Button.iButtonId := cButtonManual;
evPanelButtonRegisterData.Button.pbActionVar1 := @sv_bButtonManual;
evPanelButtonRegisterData.Button.Optional.pbLedVar := @sv_bHMILedManual;
evPanelButtonRegisterData.Button.Optional.piLedVarAttr := @sv_bHMILedManual_ledAttr;
SET_EVENT(evPanelButtonRegister, evPanelButtonRegisterData);

// register setup button
evPanelButtonRegisterData.Button.nPanelButtonType := nPanelButtonAction;
evPanelButtonRegisterData.Button.iCompId := sv_DeviceId.CompId;
evPanelButtonRegisterData.Button.iIndexId := sv_DeviceId.IndexId;
evPanelButtonRegisterData.Button.iButtonId := cButtonSetup;
evPanelButtonRegisterData.Button.pbActionVar1 := @sv_bButtonSetup;
evPanelButtonRegisterData.Button.Optional.pbLedVar := @sv_bHMILedSetup;
evPanelButtonRegisterData.Button.Optional.piLedVarAttr := @sv_bHMILedSetup_ledAttr;
SET_EVENT(evPanelButtonRegister, evPanelButtonRegisterData);

// register half-auto button
evPanelButtonRegisterData.Button.nPanelButtonType := nPanelButtonAction;
evPanelButtonRegisterData.Button.iCompId := sv_DeviceId.CompId;
evPanelButtonRegisterData.Button.iIndexId := sv_DeviceId.IndexId;
evPanelButtonRegisterData.Button.iButtonId := cButtonHalfAuto;
evPanelButtonRegisterData.Button.pbActionVar1 := @sv_bButtonHalfAuto;
evPanelButtonRegisterData.Button.Optional.pbLedVar := @sv_bHMILedHalfAutomatic;
evPanelButtonRegisterData.Button.Optional.piLedVarAttr := @sv_bHMILedHalfAutomatic_ledAttr;
SET_EVENT(evPanelButtonRegister, evPanelButtonRegisterData);

// register full-auto button
evPanelButtonRegisterData.Button.nPanelButtonType := nPanelButtonAction;
evPanelButtonRegisterData.Button.iCompId := sv_DeviceId.CompId;
evPanelButtonRegisterData.Button.iIndexId := sv_DeviceId.IndexId;
evPanelButtonRegisterData.Button.iButtonId := cButtonFullAuto;
evPanelButtonRegisterData.Button.pbActionVar1 := @sv_bButtonFullAuto;
evPanelButtonRegisterData.Button.Optional.pbLedVar := @sv_bHMILedFullAutomatic;
evPanelButtonRegisterData.Button.Optional.piLedVarAttr := @sv_bHMILedFullAutomatic_ledAttr;
SET_EVENT(evPanelButtonRegister, evPanelButtonRegisterData);

@END_Body

@@@BEG_Comment@@@
@TL(0)

@@@END_Comment@@@

@BEG_Body
@TL(39)
(**************************************** WARNING ********************************************
 *** The KEBA Kemro K2 System including software is not intended for safety control tasks! ***
 ***                       For further information see Comment tab!                        ***
 *********************************************************************************************)

//set demanded operation mode according the pressed button

bButtonManual := sv_bButtonManual;
bButtonSetup := sv_bButtonSetup;
bButtonHalfAuto := sv_bButtonHalfAuto;
bButtonFullAuto := sv_bButtonFullAuto;

IF mbDIButtonManualLinked THEN
    bButtonManual := bButtonManual OR di_ButtonManual;
END_IF;

IF mbDIButtonSetupLinked THEN
    bButtonSetup := bButtonSetup OR di_ButtonSetup;
END_IF;

IF mbDIButtonHalfAutoLinked THEN
    bButtonHalfAuto := bButtonHalfAuto OR di_ButtonHalfAuto;
END_IF;

IF mbDIButtonFullAutoLinked THEN
    bButtonFullAuto := bButtonFullAuto OR di_ButtonFullAuto;
END_IF;

IF bButtonSetup THEN
    sv_DemandedOperationMode := nSetup;
ELSIF bButtonManual THEN
    sv_DemandedOperationMode := nManual;
ELSIF bButtonHalfAuto THEN
    sv_DemandedOperationMode := nHalfAutomatic;
ELSIF bButtonFullAuto THEN
    sv_DemandedOperationMode := nFullAutomatic;
END_IF;

@END_Body

@@@BEG_Comment@@@
@TL(0)

@@@END_Comment@@@

@BEG_Body
@TL(74)
(**************************************** WARNING ********************************************
 *** The KEBA Kemro K2 System including software is not intended for safety control tasks! ***
 ***                       For further information see Comment tab!                        ***
 *********************************************************************************************)

IF sv_DemandedOperationMode = sv_OperationMode THEN
    //don´t execute if operation mode is equal demanded operation mode
    RETURN;
END_IF;

IF sv_TraceLevel.bODCInterpreter THEN
   //trace demanded opmode switch
   IF sv_DemandedOperationMode = nSetup THEN
      sDemandedOperationMode := 'Setup';
   ELSIF sv_DemandedOperationMode = nManual THEN
      sDemandedOperationMode := 'Manual';
   ELSIF sv_DemandedOperationMode = nHalfAutomatic THEN
      sDemandedOperationMode := 'HalfAutomatic';
   ELSIF sv_DemandedOperationMode = nFullAutomatic THEN
      sDemandedOperationMode := 'FullAutomatic';
   ELSE
      sDemandedOperationMode := '???';
   END_IF;
   fbDebugTrace(CONCAT('sv_DemandedOperationMode changed to ', sDemandedOperationMode));
END_IF;

IF sv_DemandedOperationMode = nFullAutomatic AND NOT sv_bAllowFullAutoMode THEN
    //change to full auto mode not allowed
    SET_ALARM (Name := erFullAutoNotAllowed);
    sv_DemandedOperationMode := sv_OperationMode;
    IF sv_TraceLevel.bODCInterpreter THEN
        fbDebugTrace('operation mode switch denied by sv_bAllowFullAutoMode');
    END_IF;
    RETURN;
END_IF;

// if demanded mode (half)automatic check if data loading is active
IF (sv_DemandedOperationMode > nManual) THEN
    IF ((sv_DataState = nReadMoldData)
        OR (sv_DataState = nReadMachineData)
        OR (sv_DataState = nReadSequenceData)
        OR (sv_DataState = nReadMaterialData)) THEN
        SET_ALARM(erAutoNotAllowed);
        sv_DemandedOperationMode := sv_OperationMode;
        IF sv_TraceLevel.bODCInterpreter THEN
            fbDebugTrace('operation mode switch denied by data loading');
        END_IF;
        RETURN;
    END_IF;
    IF (sv_LockOperationModeAuto.iLockCounter > 0) THEN
        SET_ALARM(erAutoNotAllowed);
        sv_DemandedOperationMode := sv_OperationMode;
        IF sv_TraceLevel.bODCInterpreter THEN
            fbDebugTrace('operation mode switch denied by data sv_LockOperationModeAuto');
        END_IF;
        RETURN;
    END_IF;
END_IF;

//check if demanded operation mode is allowed
abOpModeControl.aCheck(nDemandedMode := sv_DemandedOperationMode,
                       nActualMode := sv_OperationMode);

IF abOpModeControl.aCheck.bChangeAllowed THEN
    //change allowed
    sv_OperationMode := sv_DemandedOperationMode;
ELSE
    //change not allowed
    sv_DemandedOperationMode := sv_OperationMode;
    IF sv_TraceLevel.bODCInterpreter THEN
        fbDebugTrace('operation mode switch denied by abOpModeControl.aCheck()');
    END_IF;
END_IF;

@END_Body

@@@BEG_Comment@@@
@TL(0)

@@@END_Comment@@@

@BEG_Body
@TL(86)
(**************************************** WARNING ********************************************
 *** The KEBA Kemro K2 System including software is not intended for safety control tasks! ***
 ***                       For further information see Comment tab!                        ***
 *********************************************************************************************)

IF NOT bInitDone THEN
   //set HMI button led system variables
   sv_bHMILedSetup_ledAttr := 16#1;
   sv_bHMILedManual_ledAttr := 16#1;
   sv_bHMILedHalfAutomatic_ledAttr := 16#1;
   sv_bHMILedFullAutomatic_ledAttr := 16#1;

   mbLedSetupLinked := IS_LINKED(sv_bLedSetup);
   mbLedManualLinked := IS_LINKED(sv_bLedManual);
   mbLedHalfAutomaticLinked := IS_LINKED(sv_bLedHalfAutomatic);
   mbLedFullAutomaticLinked := IS_LINKED(sv_bLedFullAutomatic);

   //set led attributes
   IF IS_LINKED(sv_bLedSetup_ledAttr) THEN
      sv_bLedSetup_ledAttr := sv_bHMILedSetup_ledAttr;
      mbLedSetupAttrLinked := TRUE;
   END_IF;

   IF IS_LINKED(sv_bLedManual_ledAttr) THEN
      sv_bLedManual_ledAttr := sv_bHMILedManual_ledAttr;
      mbLedManualAttrLinked := TRUE;
   END_IF;

   IF IS_LINKED(sv_bLedHalfAutomatic_ledAttr) THEN
      sv_bLedHalfAutomatic_ledAttr := sv_bHMILedHalfAutomatic_ledAttr;
      mbLedHalfAutomaticAttrLinked := TRUE;
   END_IF;

   IF IS_LINKED(sv_bLedFullAutomatic_ledAttr) THEN
      sv_bLedFullAutomatic_ledAttr := sv_bHMILedFullAutomatic_ledAttr;
      mbLedFullAutomaticAttrLinked := TRUE;
   END_IF;

   bInitDone := TRUE;
END_IF;

IF (sv_OperationMode = nManual) THEN
   sv_bHMILedManual := TRUE;
   sv_bHMILedSetup := FALSE;
   sv_bHMILedHalfAutomatic := FALSE;
   sv_bHMILedFullAutomatic := FALSE;

ELSIF (sv_OperationMode = nSetup) THEN
   sv_bHMILedManual := FALSE;
   sv_bHMILedSetup := TRUE;
   sv_bHMILedHalfAutomatic := FALSE;
   sv_bHMILedFullAutomatic := FALSE;

ELSIF (sv_OperationMode = nHalfAutomatic) THEN
   sv_bHMILedManual := FALSE;
   sv_bHMILedSetup := FALSE;
   sv_bHMILedHalfAutomatic := TRUE;
   sv_bHMILedFullAutomatic := FALSE;

ELSIF (sv_OperationMode = nFullAutomatic) THEN
   sv_bHMILedManual := FALSE;
   sv_bHMILedSetup := FALSE;
   sv_bHMILedHalfAutomatic := FALSE;
   sv_bHMILedFullAutomatic := TRUE;

END_IF;

// copy the led states to the hw-leds
IF mbLedSetupLinked THEN
   sv_bLedSetup := sv_bHMILedSetup;
END_IF;

IF mbLedManualLinked THEN
   sv_bLedManual := sv_bHMILedManual;
END_IF;

IF mbLedHalfAutomaticLinked THEN
   sv_bLedHalfAutomatic := sv_bHMILedHalfAutomatic;
END_IF;

IF mbLedFullAutomaticLinked THEN
   sv_bLedFullAutomatic := sv_bHMILedFullAutomatic;
END_IF;

@END_Body

@@@BEG_Comment@@@
@TL(0)

@@@END_Comment@@@

@BEG_Body
@TL(14)
(**************************************** WARNING ********************************************
 *** The KEBA Kemro K2 System including software is not intended for safety control tasks! ***
 ***                       For further information see Comment tab!                        ***
 *********************************************************************************************)

//do not change mode if operation mode is already manual or setup
IF sv_OperationMode >= nHalfAutomatic THEN
   IF sv_TraceLevel.bODCInterpreter THEN
      fbDebugTrace(CONCAT('switching opmode to manual because of evAlarmAutoManual (',
                          GET_ALARM_NAME(evAlarmAutoManualData.NAME), ')'));
   END_IF;
   sv_DemandedOperationMode := nManual;
END_IF;

@END_Body

@@@BEG_Comment@@@
@TL(0)

@@@END_Comment@@@

@BEG_Body
@TL(14)
(**************************************** WARNING ********************************************
 *** The KEBA Kemro K2 System including software is not intended for safety control tasks! ***
 ***                       For further information see Comment tab!                        ***
 *********************************************************************************************)

//do not change mode if operation mode is already not full auto
IF sv_OperationMode = nFullAutomatic THEN
   IF sv_TraceLevel.bODCInterpreter THEN
      fbDebugTrace(CONCAT('switching opmode to half auto because of evAlarmAutoHalf (',
                          GET_ALARM_NAME(evAlarmAutoManualData.NAME), ')'));
   END_IF;
   sv_DemandedOperationMode := nHalfAutomatic;
END_IF;

@END_Body

@@@BEG_Comment@@@
@TL(0)

@@@END_Comment@@@

@BEG_Body
@TL(23)
(**************************************** WARNING ********************************************
 *** The KEBA Kemro K2 System including software is not intended for safety control tasks! ***
 ***                       For further information see Comment tab!                        ***
 *********************************************************************************************)

IF (sv_OperationMode <> nSetup) THEN
   IF sv_bOverrideCoreSafety THEN
      //reset override core safety flag if mode is not setup mode
      //and set alarm
      sv_bOverrideCoreSafety := FALSE;
      SET_ALARM(erSetupModeRequired);
   END_IF;

   IF sv_bOverrideEjectorSafety THEN
      //reset override ejector safety flag if mode is not setup mode
      //and set alarm
      sv_bOverrideEjectorSafety := FALSE;
      SET_ALARM(erSetupModeRequired);
   END_IF;
END_IF;

@END_Body

@@@BEG_Comment@@@
@TL(0)

@@@END_Comment@@@

@BEG_Body
@TL(11)
(**************************************** WARNING ********************************************
 *** The KEBA Kemro K2 System including software is not intended for safety control tasks! ***
 ***                       For further information see Comment tab!                        ***
 *********************************************************************************************)

IF sv_OperationMode <> nSetup THEN
   //reset "override safety" flags if setup mode is left
   sv_bOverrideCoreSafety := FALSE;
   sv_bOverrideEjectorSafety := FALSE;
END_IF;

@END_Body

@@@BEG_Comment@@@
@TL(0)

@@@END_Comment@@@
@END_Body

@END_Contents

(* ---- ABOperationModeLockManager.pu ---- *)
IMPORT_OVER_LISTFILE
 ABResourceLockManager
, tsLockOperationModeAuto
, tsResourceLock

END_IMPORT

ALGORITHM_BLOCK ABOperationModeLockManager #DUMMY_EDIT_BLOCK

SYSTEM_VAR
 sv_LockOperationModeAuto : tsLockOperationModeAuto;
 sv_LockDataState : tsResourceLock;
END_VAR

SYSTEM_OBJECT
 TaskSlow : TASK;
END_OBJECT

VAR
 abModeAutoLockManager : ABResourceLockManager;
 abDataStateLockManager : ABResourceLockManager;
END_VAR

PROCESS_ALGORITHM paInit ON TaskSlow AUTOSTART

#BEGIN_EDIT_BLOCK
abModeAutoLockManager.aInit("LockOpModeAuto", @sv_LockOperationModeAuto.sResourceLock, T#10s);
abDataStateLockManager.aInit("LockDataState", @sv_LockDataState, T#3m);
STOP_PROCESS_ALGORITHM();

;#END_EDIT_BLOCK END_ALGORITHM

END_ALGORITHM_BLOCK

#END_OF_IEC_PART

@Puma @IecEditor 6 159 @Pou 25
@@@BEG_Comment@@@

@@@END_Comment@@@

@BEG_Contents

@BEG_Func
@RT(17)FuncTreeContainer
0
@END_Func

@BEG_Const
@RT(18)ConstTreeContainer
0
@END_Const

@BEG_Export

@BEG_Kind
@ALGORITHM_BLOCK @RT(26)ABOperationModeLockManager @STRUCTURED_TEXT
@RT(0) @RT(0) @RT(0)
@END_Kind

@BEG_Dcl
@RT(16)DclTreeContainer
5
@Var @RT(21)abModeAutoLockManager @RT(0) @T @T @DERIVED 0 @T @T @DT @RT(21)ABResourceLockManager @RT(0) @T @T @UNKNOWN 0 @F
@F @F
@T
@BEG_Attrib
3 @RT(0) @RT(0) @RT(0)
@END_Attrib
1 0 @F @F @F @F

@Var @RT(22)abDataStateLockManager @RT(0) @T @T @DERIVED 0 @T @T @DT @RT(21)ABResourceLockManager @RT(0) @T @T @UNKNOWN 0 @F
@F @F
@T
@BEG_Attrib
3 @RT(0) @RT(0) @RT(0)
@END_Attrib
1 0 @F @F @F @F

@Var @RT(24)sv_LockOperationModeAuto @RT(0) @T @T @DERIVED 0 @T @T @DT @RT(23)tsLockOperationModeAuto @RT(0) @T @T @UNKNOWN 0 @F
@F @F
@T
@BEG_Attrib
3 @RT(0) @RT(0) @RT(0)
@END_Attrib
1 8 @F @F @F @F

@Var @RT(16)sv_LockDataState @RT(0) @T @T @DERIVED 0 @T @T @DT @RT(14)tsResourceLock @RT(0) @T @T @UNKNOWN 0 @F
@F @F
@T
@BEG_Attrib
3 @RT(0) @RT(0) @RT(0)
@END_Attrib
1 8 @F @F @F @F

@Var @RT(8)TaskSlow @RT(0) @T @T @RENAMED 0 @T @T @DT @RT(4)TASK @RT(0) @T @T @BASIC 0 @F
@F @F
@T
@BEG_Attrib
3 @RT(0) @RT(0) @RT(0)
@END_Attrib
1 7 @F @F @F @F

@END_Dcl

@END_Export

@BEG_Body

1

@BEG_Export

@BEG_Algo
@PROCESS_ALGORITHM @RT(6)paInit @STRUCTURED_TEXT
@RT(0) @RT(0) @RT(8)TaskSlow @T @F
@END_Algo

@BEG_Dcl
@RT(16)DclTreeContainer
0
@END_Dcl

@END_Export

@BEG_Body
@TL(4)
abModeAutoLockManager.aInit("LockOpModeAuto", @sv_LockOperationModeAuto.sResourceLock, T#10s);
abDataStateLockManager.aInit("LockDataState", @sv_LockDataState, T#3m);
STOP_PROCESS_ALGORITHM();

@END_Body

@@@BEG_Comment@@@
@TL(0)

@@@END_Comment@@@
@END_Body

@END_Contents

(* ---- ABOpModeControl.pu ---- *)
IMPORT_OVER_LISTFILE
 cCompAll
, cModeAutomatic
, cModeFullAutomatic
, tevLockUnlock
, tsTraceLevel
, tsActiveMovements
, tsDeviceId
, tnSafetyGateState
, tsMoveCtrl
, ABLockList
, FBDebugTrace
, tevLockUnlockData
, tnOperationMode

END_IMPORT

ALGORITHM_BLOCK ABOpModeControl #DUMMY_EDIT_BLOCK

SYSTEM_VAR
 sv_TraceLevel : tsTraceLevel;
 sv_ActiveMovements : tsActiveMovements;
 sv_DeviceId : tsDeviceId;
 sv_iPendingAlarms : DINT;
 sv_MoldSafetyGateState : tnSafetyGateState;
END_VAR

SYSTEM_OBJECT
 EV_Task_3 : TASK;
 evLockUnlock : tevLockUnlock;
END_OBJECT

VAR_EXTERNAL
 g_MoveCtrl : tsMoveCtrl;
END_VAR

VAR
 abLockList : ABLockList;
 fbDebugTrace : FBDebugTrace;
END_VAR

EVENT_ALGORITHM evaLockUnlock ON EV_Task_3 WITH evLockUnlock

VAR_INPUT
 evLockUnlockData : tevLockUnlockData;
END_VAR
#BEGIN_EDIT_BLOCK
(**************************************** WARNING ********************************************
 *** The KEBA Kemro K2 System including software is not intended for safety control tasks! ***
 ***                       For further information see Comment tab!                        ***
 *********************************************************************************************)

IF (evLockUnlockData.DeviceId.CompId = sv_DeviceId.CompId   OR evLockUnlockData.DeviceId.CompId =  cCompAll    ) AND
   (evLockUnlockData.DeviceId.IndexId = sv_DeviceId.IndexId OR evLockUnlockData.DeviceId.IndexId = cAllDevIndex) THEN

      IF evLockUnlockData.Mode = nUnlock THEN
         // UNLOCK Movement
         g_MoveCtrl.bStop := FALSE;
         abLockList.aRemove.Entry.DeviceIdSender := evLockUnlockData.DeviceIdSender;
         abLockList.aRemove.Entry.MoveDir        := evLockUnlockData.MoveDir;
         abLockList.aRemove.Entry.MoveId         := evLockUnlockData.MoveId;
         abLockList.aRemove.Entry.Alarm          := evLockUnlockData.Alarm;
         // remove movement from locklist
         abLockList.aRemove();

         IF sv_TraceLevel.bLockUnlock THEN
            fbDebugTrace(CONCAT("movement ",
                                DINT_TO_STRING(evLockUnlockData.MoveDir), '/', DINT_TO_STRING(evLockUnlockData.MoveId),
                                ' unlocked by Device: ',
                                DINT_TO_STRING(evLockUnlockData.DeviceIdSender.CompId), '.', DINT_TO_STRING(evLockUnlockData.DeviceIdSender.IndexId),
                                ' alarm ', GET_ALARM_NAME(evLockUnlockData.Alarm.AlarmId)));
         END_IF;
      ELSE
         // LOCK Movement
         abLockList.aAdd.Entry.DeviceIdSender   := evLockUnlockData.DeviceIdSender;
         abLockList.aAdd.Entry.MoveDir          := evLockUnlockData.MoveDir;
         abLockList.aAdd.Entry.MoveId           := evLockUnlockData.MoveId;
         abLockList.aAdd.Entry.Alarm            := evLockUnlockData.Alarm;
         abLockList.aAdd.bDisable               := FALSE;

         IF evLockUnlockData.Mode = nLockResume THEN

            abLockList.aAdd.Entry.bStopDevice := FALSE;

         ELSIF evLockUnlockData.Mode = nLockAbort THEN

            abLockList.aAdd.Entry.bStopDevice := TRUE;
         END_IF;

         abLockList.aAdd.bSetAlarmImmediately := evLockUnlockData.bSetAlarmImmediately;

         // add movement to locklist
         abLockList.aAdd();

         IF sv_TraceLevel.bLockUnlock THEN
            fbDebugTrace(CONCAT("movement ",
                                DINT_TO_STRING(evLockUnlockData.MoveDir), '/', DINT_TO_STRING(evLockUnlockData.MoveId),
                                ' locked   by Device: ',
                                DINT_TO_STRING(evLockUnlockData.DeviceIdSender.CompId), '.', DINT_TO_STRING(evLockUnlockData.DeviceIdSender.IndexId),
                                ' alarm ', GET_ALARM_NAME(evLockUnlockData.Alarm.AlarmId)));
         END_IF;
      END_IF;

END_IF;

;#END_EDIT_BLOCK END_ALGORITHM

ALGORITHM aCheck

VAR_INPUT
 nActualMode : tnOperationMode (* actual operation mode *);
 nDemandedMode : tnOperationMode (* demanded operation mode *);
END_VAR

VAR_OUTPUT
 bChangeAllowed : BOOL (* change to demanded mode is allowed *);
END_VAR

VAR
 bAllow : BOOL;
 iActiveMoves : DINT;
 bHalfAutoLocked : BOOL;
 bFullAutoLocked : BOOL;
 bPendingAlarmsOk : BOOL;
END_VAR

(* IecGraph-Code *)

(* init step *)
INITIAL_STEP S_Init:
AInit (P);
END_STEP

ACTION AInit: #BEGIN_EDIT_BLOCK
bAllow := FALSE;

;#END_EDIT_BLOCK END_ACTION (*AInit*)

(* steps *)
STEP S_CheckActualMode:
END_STEP

STEP S_FullAuto:
AFullAuto (P);
END_STEP

ACTION AFullAuto: #BEGIN_EDIT_BLOCK
bAllow := TRUE;

;#END_EDIT_BLOCK END_ACTION (*AFullAuto*)
STEP S_CheckDemandedMode:
END_STEP

STEP S_FullAutoDemanded:
ACheck (P);
END_STEP

STEP S_ModeAllowed:
AChangeAllowed (P);
END_STEP

ACTION AChangeAllowed: #BEGIN_EDIT_BLOCK
bAllow := TRUE;

;#END_EDIT_BLOCK END_ACTION (*AChangeAllowed*)
STEP S_CheckActiveMoves:
AGetActiveMovements (P);
END_STEP

ACTION AGetActiveMovements: #BEGIN_EDIT_BLOCK
iActiveMoves := sv_ActiveMovements.iNumberOfActiveMovements;

;#END_EDIT_BLOCK END_ACTION (*AGetActiveMovements*)
STEP S_CheckDemand:
END_STEP

STEP S_AllowMode:
AAllowedMode (P);
END_STEP

ACTION AAllowedMode: #BEGIN_EDIT_BLOCK
bAllow := TRUE;

;#END_EDIT_BLOCK END_ACTION (*AAllowedMode*)
STEP S_CheckAlarms:
ACheckPendingAlarms (P);
END_STEP

STEP S_CheckAutoAllowed:
Action15 (P);
END_STEP

STEP S_End:
ACopyResult (P);
END_STEP

ACTION ACopyResult: #BEGIN_EDIT_BLOCK
bChangeAllowed := bAllow;

;#END_EDIT_BLOCK END_ACTION (*ACopyResult*)

(* transitions *)
GO_ON_TRANSITION TInitDone (* Trans6 *) FROM S_Init TO S_CheckActualMode :=  #BEGIN_EDIT_BLOCK
TRUE
;#END_EDIT_BLOCK
END_TRANSITION

GO_ON_TRANSITION TFullAuto (* Trans1 *) FROM S_CheckActualMode TO S_FullAuto :=  #BEGIN_EDIT_BLOCK
nActualMode = nFullAutomatic
;#END_EDIT_BLOCK
END_TRANSITION

GO_ON_TRANSITION Trans5 (* Trans5 *) FROM S_FullAuto TO S_End :=  #BEGIN_EDIT_BLOCK
TRUE
;#END_EDIT_BLOCK
END_TRANSITION

GO_ON_TRANSITION THalfAuto (* Trans2 *) FROM S_CheckActualMode TO S_CheckDemandedMode :=  #BEGIN_EDIT_BLOCK
nActualMode = nHalfAutomatic
;#END_EDIT_BLOCK
END_TRANSITION

GO_ON_TRANSITION TDemandFullAuto (* Trans8 *) FROM S_CheckDemandedMode TO S_FullAutoDemanded :=  #BEGIN_EDIT_BLOCK
nDemandedMode = nFullAutomatic
;#END_EDIT_BLOCK
END_TRANSITION

GO_ON_TRANSITION Trans11 (* Trans11 *) FROM S_FullAutoDemanded TO S_End :=  #BEGIN_EDIT_BLOCK
TRUE
;#END_EDIT_BLOCK
END_TRANSITION

GO_ON_TRANSITION TDemandManualOrSetup (* Trans9 *) FROM S_CheckDemandedMode TO S_ModeAllowed :=  #BEGIN_EDIT_BLOCK
nDemandedMode <> nFullAutomatic
;#END_EDIT_BLOCK
END_TRANSITION

GO_ON_TRANSITION Trans10 (* Trans10 *) FROM S_ModeAllowed TO S_End :=  #BEGIN_EDIT_BLOCK
TRUE
;#END_EDIT_BLOCK
END_TRANSITION

GO_ON_TRANSITION TSetupOrManual (* Trans3 *) FROM S_CheckActualMode TO S_CheckActiveMoves :=  #BEGIN_EDIT_BLOCK
nActualMode = nSetup OR nActualMode = nManual
;#END_EDIT_BLOCK
END_TRANSITION

GO_ON_TRANSITION TNoMovesActive (* Trans12 *) FROM S_CheckActiveMoves TO S_CheckDemand :=  #BEGIN_EDIT_BLOCK
iActiveMoves = 0
;#END_EDIT_BLOCK
END_TRANSITION

GO_ON_TRANSITION TMovesActive (* Trans25 *) FROM S_CheckActiveMoves TO S_End :=  #BEGIN_EDIT_BLOCK
iActiveMoves > 0
;#END_EDIT_BLOCK
END_TRANSITION

GO_ON_TRANSITION TLowerHalfAuto (* Trans15 *) FROM S_CheckDemand TO S_AllowMode :=  #BEGIN_EDIT_BLOCK
nDemandedMode < nHalfAutomatic
;#END_EDIT_BLOCK
END_TRANSITION

GO_ON_TRANSITION Trans16 (* Trans16 *) FROM S_AllowMode TO S_End :=  #BEGIN_EDIT_BLOCK
TRUE
;#END_EDIT_BLOCK
END_TRANSITION

GO_ON_TRANSITION TAutoModeDemanded (* Trans17 *) FROM S_CheckDemand TO S_CheckAlarms :=  #BEGIN_EDIT_BLOCK
nDemandedMode > nManual
;#END_EDIT_BLOCK
END_TRANSITION

GO_ON_TRANSITION TNoActiveAlarms (* Trans20 *) FROM S_CheckAlarms TO S_CheckAutoAllowed :=  #BEGIN_EDIT_BLOCK
bPendingAlarmsOk
;#END_EDIT_BLOCK
END_TRANSITION

GO_ON_TRANSITION TAcitveAlarms (* Trans24 *) FROM S_CheckAlarms TO S_End :=  #BEGIN_EDIT_BLOCK
NOT bPendingAlarmsOk
;#END_EDIT_BLOCK
END_TRANSITION

GO_ON_TRANSITION Trans18 (* Trans18 *) FROM S_CheckAutoAllowed TO S_End :=  #BEGIN_EDIT_BLOCK
TRUE
;#END_EDIT_BLOCK
END_TRANSITION

TRANSITION TWaitForNextCall (* Trans19 *) FROM S_End TO S_Init :=  #BEGIN_EDIT_BLOCK
TRUE
;#END_EDIT_BLOCK
END_TRANSITION

(* end IecGraph-Code *)
(* sfc-code *)

(* stand alone actions *)
ACTION ACheck: #BEGIN_EDIT_BLOCK
// check if full auto mode is locked
abLockList.aCheck(MoveDir := cModeFullAutomatic,
                  MoveId := cModeFullAutomatic);
bAllow := NOT abLockList.aCheck.bLocked;

;#END_EDIT_BLOCK END_ACTION (*ACheck*)
ACTION Action15: #BEGIN_EDIT_BLOCK
IF nDemandedMode = nFullAutomatic THEN
    //full auto mode demanded -> check if full auto is locked
    abLockList.aCheck(MoveDir := cModeFullAutomatic,
                        MoveId := cModeFullAutomatic);
    bFullAutoLocked := abLockList.aCheck.bLocked;

    //check if half and full auto is locked
    abLockList.aCheck(MoveDir := cModeAutomatic,
                        MoveId := cModeAutomatic);
    bHalfAutoLocked := abLockList.aCheck.bLocked;

    bAllow := NOT bHalfAutoLocked AND NOT bFullAutoLocked;
ELSIF nDemandedMode = nHalfAutomatic THEN
    //half auto mode demanded
    abLockList.aCheck(MoveDir := cModeAutomatic,
                        MoveId := cModeAutomatic);
    bAllow := NOT abLockList.aCheck.bLocked;
ELSE
    bAllow := TRUE;
END_IF;

;#END_EDIT_BLOCK END_ACTION (*Action15*)
ACTION ACheckPendingAlarms: #BEGIN_EDIT_BLOCK
(**************************************** WARNING ********************************************
 *** The KEBA Kemro K2 System including software is not intended for safety control tasks! ***
 ***                       For further information see Comment tab!                        ***
 *********************************************************************************************)

//basically operation mode can not be changed to HA or FA if any alarm of class 1, 2 or 3 is pending
//there is only one exception:
//If the mold safety gate is open it should also be possible to switch to HA and FA
bPendingAlarmsOk := (sv_iPendingAlarms = 0) OR ((sv_iPendingAlarms = 1) AND (sv_MoldSafetyGateState = nOpen));

;#END_EDIT_BLOCK END_ACTION (*ACheckPendingAlarms*)
(* end sfc-code *)

END_ALGORITHM

END_ALGORITHM_BLOCK

#END_OF_IEC_PART

@Puma @IecEditor 6 68 @Pou 25
@@@BEG_Comment@@@

@@@END_Comment@@@

@BEG_Contents

@BEG_Func
@RT(17)FuncTreeContainer
0
@END_Func

@BEG_Const
@RT(18)ConstTreeContainer
3
@Var @RT(8)cCompAll @RT(0) @T @F @DT @RT(4)DINT @RT(0) @T @T @BASIC 0 @F
@F @F
@T
@BEG_Attrib
0 @RT(10)cMaxCompId @RT(22)to lock all components
@END_Attrib
1 1 @F @F @F @F

@Var @RT(14)cModeAutomatic @RT(0) @T @F @DT @RT(4)DINT @RT(0) @T @T @BASIC 0 @F
@F @F
@T
@BEG_Attrib
0 @RT(2)23 @RT(50)for locking/unlocking half and full automatic mode
@END_Attrib
1 1 @F @F @F @F

@Var @RT(18)cModeFullAutomatic @RT(0) @T @F @DT @RT(4)DINT @RT(0) @T @T @BASIC 0 @F
@F @F
@T
@BEG_Attrib
0 @RT(2)24 @RT(46)for locking/unlocking only full automatic mode
@END_Attrib
1 1 @F @F @F @F

@END_Const

@BEG_Export

@BEG_Kind
@ALGORITHM_BLOCK @RT(15)ABOpModeControl @STRUCTURED_TEXT
@RT(0) @RT(0) @RT(0)
@END_Kind

@BEG_Dcl
@RT(16)DclTreeContainer
10
@Var @RT(9)EV_Task_3 @RT(0) @T @F @DT @RT(4)TASK @RT(0) @T @T @BASIC 0 @F
@F @F
@T
@BEG_Attrib
3 @RT(0) @RT(0) @RT(0)
@END_Attrib
1 7 @F @F @F @F

@Var @RT(12)evLockUnlock @RT(0) @T @T @DERIVED 0 @T @T @DT @RT(13)tevLockUnlock @RT(0) @T @T @UNKNOWN 0 @F
@F @F
@T
@BEG_Attrib
3 @RT(0) @RT(0) @RT(0)
@END_Attrib
1 7 @F @F @F @F

@Var @RT(13)sv_TraceLevel @RT(0) @T @T @RENAMED 0 @T @T @DT @RT(12)tsTraceLevel @RT(0) @T @T @UNKNOWN 0 @F
@F @F
@T
@BEG_Attrib
3 @RT(0) @RT(0) @RT(0)
@END_Attrib
1 8 @F @F @F @F

@Var @RT(18)sv_ActiveMovements @RT(0) @T @T @DERIVED 0 @T @T @DT @RT(17)tsActiveMovements @RT(0) @T @T @UNKNOWN 0 @F
@F @F
@T
@BEG_Attrib
3 @RT(0) @RT(0) @RT(0)
@END_Attrib
1 8 @F @F @F @F

@Var @RT(11)sv_DeviceId @RT(0) @T @T @DERIVED 0 @T @T @DT @RT(10)tsDeviceId @RT(0) @T @T @UNKNOWN 0 @F
@F @F
@T
@BEG_Attrib
3 @RT(0) @RT(0) @RT(0)
@END_Attrib
1 8 @F @F @F @F

@Var @RT(17)sv_iPendingAlarms @RT(0) @T @F @DT @RT(4)DINT @RT(0) @T @T @BASIC 0 @F
@F @F
@T
@BEG_Attrib
3 @RT(0) @RT(0) @RT(0)
@END_Attrib
1 8 @F @F @F @F

@Var @RT(22)sv_MoldSafetyGateState @RT(0) @T @T @DERIVED 0 @T @T @DT @RT(17)tnSafetyGateState @RT(0) @T @T @UNKNOWN 0 @F
@F @F
@T
@BEG_Attrib
3 @RT(0) @RT(0) @RT(0)
@END_Attrib
1 8 @F @F @F @F

@Var @RT(10)g_MoveCtrl @RT(0) @T @T @DERIVED 0 @T @T @DT @RT(10)tsMoveCtrl @RT(0) @T @T @UNKNOWN 0 @F
@F @F
@T
@BEG_Attrib
3 @RT(0) @RT(0) @RT(0)
@END_Attrib
1 6 @F @F @F @F

@Var @RT(10)abLockList @RT(0) @T @T @DERIVED 0 @F @RT(10)ABLockList @F
@T
@BEG_Attrib
3 @RT(0) @RT(0) @RT(0)
@END_Attrib
1 0 @F @F @F @F

@Var @RT(12)fbDebugTrace @RT(0) @T @T @DERIVED 0 @T @T @DT @RT(12)FBDebugTrace @RT(0) @T @T @UNKNOWN 0 @F
@F @F
@T
@BEG_Attrib
3 @RT(0) @RT(0) @RT(0)
@END_Attrib
1 0 @F @F @F @F

@END_Dcl

@END_Export

@BEG_Body

2

@BEG_Export

@BEG_Algo
@EVENT_ALGORITHM @RT(13)evaLockUnlock @STRUCTURED_TEXT
@RT(0) @RT(12)evLockUnlock @RT(9)EV_Task_3 @F @F
@END_Algo

@BEG_Dcl
@RT(16)DclTreeContainer
1
@Var @RT(16)evLockUnlockData @RT(0) @T @T @DERIVED 0 @T @T @DT @RT(17)tevLockUnlockData @RT(0) @T @T @UNKNOWN 0 @F
@F @F
@T
@BEG_Attrib
3 @RT(0) @RT(0) @RT(0)
@END_Attrib
1 1 @F @F @F @F

@END_Dcl

@END_Export

@BEG_Export

@BEG_Algo
@ALGORITHM @RT(6)aCheck @SEQUENTIAL_FLOW_CHART
@RT(0) @RT(0) @RT(0) @F @F
@END_Algo

@BEG_Dcl
@RT(16)DclTreeContainer
8
@Var @RT(11)nActualMode @RT(0) @T @T @DERIVED 0 @T @T @DT @RT(15)tnOperationMode @RT(0) @T @T @UNKNOWN 0 @F
@F @F
@T
@BEG_Attrib
3 @RT(0) @RT(21)actual operation mode @RT(0)
@END_Attrib
1 1 @F @F @F @F

@Var @RT(13)nDemandedMode @RT(0) @T @T @DERIVED 0 @T @T @DT @RT(15)tnOperationMode @RT(0) @T @T @UNKNOWN 0 @F
@F @F
@T
@BEG_Attrib
3 @RT(0) @RT(23)demanded operation mode @RT(0)
@END_Attrib
1 1 @F @F @F @F

@Var @RT(14)bChangeAllowed @RT(0) @T @F @DT @RT(4)BOOL @RT(0) @T @T @BASIC 0 @F
@F @F
@T
@BEG_Attrib
3 @RT(0) @RT(34)change to demanded mode is allowed @RT(0)
@END_Attrib
1 3 @F @F @F @F

@Var @RT(6)bAllow @RT(0) @T @F @DT @RT(4)BOOL @RT(0) @T @T @BASIC 0 @F
@F @F
@T
@BEG_Attrib
3 @RT(0) @RT(0) @RT(0)
@END_Attrib
1 0 @F @F @F @F

@Var @RT(12)iActiveMoves @RT(0) @T @F @DT @RT(4)DINT @RT(0) @T @T @BASIC 0 @F
@F @F
@T
@BEG_Attrib
3 @RT(0) @RT(0) @RT(0)
@END_Attrib
1 0 @F @F @F @F

@Var @RT(15)bHalfAutoLocked @RT(0) @T @F @DT @RT(4)BOOL @RT(0) @T @T @BASIC 0 @F
@F @F
@T
@BEG_Attrib
3 @RT(0) @RT(0) @RT(0)
@END_Attrib
1 0 @F @F @F @F

@Var @RT(15)bFullAutoLocked @RT(0) @T @F @DT @RT(4)BOOL @RT(0) @T @T @BASIC 0 @F
@F @F
@T
@BEG_Attrib
3 @RT(0) @RT(0) @RT(0)
@END_Attrib
1 0 @F @F @F @F

@Var @RT(16)bPendingAlarmsOk @RT(0) @T @F @DT @RT(4)BOOL @RT(0) @T @T @BASIC 0 @F
@F @F
@T
@BEG_Attrib
3 @RT(0) @RT(0) @RT(0)
@END_Attrib
1 0 @F @F @F @F

@END_Dcl

@END_Export

@BEG_Body
@TL(59)
(**************************************** WARNING ********************************************
 *** The KEBA Kemro K2 System including software is not intended for safety control tasks! ***
 ***                       For further information see Comment tab!                        ***
 *********************************************************************************************)

IF (evLockUnlockData.DeviceId.CompId = sv_DeviceId.CompId   OR evLockUnlockData.DeviceId.CompId =  cCompAll    ) AND
   (evLockUnlockData.DeviceId.IndexId = sv_DeviceId.IndexId OR evLockUnlockData.DeviceId.IndexId = cAllDevIndex) THEN

      IF evLockUnlockData.Mode = nUnlock THEN
         // UNLOCK Movement
         g_MoveCtrl.bStop := FALSE;
         abLockList.aRemove.Entry.DeviceIdSender := evLockUnlockData.DeviceIdSender;
         abLockList.aRemove.Entry.MoveDir        := evLockUnlockData.MoveDir;
         abLockList.aRemove.Entry.MoveId         := evLockUnlockData.MoveId;
         abLockList.aRemove.Entry.Alarm          := evLockUnlockData.Alarm;
         // remove movement from locklist
         abLockList.aRemove();

         IF sv_TraceLevel.bLockUnlock THEN
            fbDebugTrace(CONCAT("movement ",
                                DINT_TO_STRING(evLockUnlockData.MoveDir), '/', DINT_TO_STRING(evLockUnlockData.MoveId),
                                ' unlocked by Device: ',
                                DINT_TO_STRING(evLockUnlockData.DeviceIdSender.CompId), '.', DINT_TO_STRING(evLockUnlockData.DeviceIdSender.IndexId),
                                ' alarm ', GET_ALARM_NAME(evLockUnlockData.Alarm.AlarmId)));
         END_IF;
      ELSE
         // LOCK Movement
         abLockList.aAdd.Entry.DeviceIdSender   := evLockUnlockData.DeviceIdSender;
         abLockList.aAdd.Entry.MoveDir          := evLockUnlockData.MoveDir;
         abLockList.aAdd.Entry.MoveId           := evLockUnlockData.MoveId;
         abLockList.aAdd.Entry.Alarm            := evLockUnlockData.Alarm;
         abLockList.aAdd.bDisable               := FALSE;

         IF evLockUnlockData.Mode = nLockResume THEN

            abLockList.aAdd.Entry.bStopDevice := FALSE;

         ELSIF evLockUnlockData.Mode = nLockAbort THEN

            abLockList.aAdd.Entry.bStopDevice := TRUE;
         END_IF;

         abLockList.aAdd.bSetAlarmImmediately := evLockUnlockData.bSetAlarmImmediately;

         // add movement to locklist
         abLockList.aAdd();

         IF sv_TraceLevel.bLockUnlock THEN
            fbDebugTrace(CONCAT("movement ",
                                DINT_TO_STRING(evLockUnlockData.MoveDir), '/', DINT_TO_STRING(evLockUnlockData.MoveId),
                                ' locked   by Device: ',
                                DINT_TO_STRING(evLockUnlockData.DeviceIdSender.CompId), '.', DINT_TO_STRING(evLockUnlockData.DeviceIdSender.IndexId),
                                ' alarm ', GET_ALARM_NAME(evLockUnlockData.Alarm.AlarmId)));
         END_IF;
      END_IF;

END_IF;

@END_Body

@@@BEG_Comment@@@
@TL(0)

@@@END_Comment@@@

@BEG_SfcBody
22 18 26

@BEG_SfcData 2
@StepSeq @RT(4)sseq @F 1
@Loop @RT(4)loop @F 2
@StepSeq @RT(3)seq @F 5
@Step @RT(6)S_Init @F @T @F @F @RT(0) @F
@AcbCont @RT(7)unnamed @F 1
@Acb @RT(5)AInit @F @T @RT(1)P @RT(0) @F @F @T @TL(2)
bAllow := FALSE;

@F

@Trans @RT(9)TInitDone @F @T @F @F @T @F @TL(2)
TRUE

@RT(6)Trans6 @F
@Step @RT(17)S_CheckActualMode @F @F @F @F @RT(0) @F
@AcbCont @RT(7)unnamed @F 0

@AltBranch @RT(3)alt @F 3
@TransSeq @RT(4)tseq @F 3
@Trans @RT(9)TFullAuto @F @T @F @F @T @F @TL(2)
nActualMode = nFullAutomatic

@RT(6)Trans1 @F
@Step @RT(10)S_FullAuto @F @F @F @F @RT(0) @F
@AcbCont @RT(7)unnamed @F 1
@Acb @RT(9)AFullAuto @F @T @RT(1)P @RT(0) @F @F @T @TL(2)
bAllow := TRUE;

@F

@Trans @RT(6)Trans5 @F @T @F @F @T @F @TL(2)
TRUE

@RT(6)Trans5 @F

@TransSeq @RT(4)tseq @F 3
@Trans @RT(9)THalfAuto @F @T @F @F @T @F @TL(2)
nActualMode = nHalfAutomatic

@RT(6)Trans2 @F
@Step @RT(19)S_CheckDemandedMode @F @F @F @F @RT(0) @F
@AcbCont @RT(7)unnamed @F 0

@AltBranch @RT(3)alt @F 2
@TransSeq @RT(4)tseq @F 3
@Trans @RT(15)TDemandFullAuto @F @T @F @F @T @F @TL(2)
nDemandedMode = nFullAutomatic

@RT(6)Trans8 @F
@Step @RT(18)S_FullAutoDemanded @F @F @F @F @RT(0) @F
@AcbCont @RT(7)unnamed @F 1
@Acb @RT(6)ACheck @F @F @RT(1)P @RT(0) @F @F @F @F

@Trans @RT(7)Trans11 @F @T @F @F @T @F @TL(2)
TRUE

@RT(7)Trans11 @F

@TransSeq @RT(4)tseq @F 3
@Trans @RT(20)TDemandManualOrSetup @F @T @F @F @T @F @TL(2)
nDemandedMode <> nFullAutomatic

@RT(6)Trans9 @F
@Step @RT(13)S_ModeAllowed @F @F @F @F @RT(0) @F
@AcbCont @RT(7)unnamed @F 1
@Acb @RT(14)AChangeAllowed @F @T @RT(1)P @RT(0) @F @F @T @TL(2)
bAllow := TRUE;

@F

@Trans @RT(7)Trans10 @F @T @F @F @T @F @TL(2)
TRUE

@RT(7)Trans10 @F

@TransSeq @RT(4)tseq @F 5
@Trans @RT(14)TSetupOrManual @F @T @F @F @T @F @TL(2)
nActualMode = nSetup OR nActualMode = nManual

@RT(6)Trans3 @F
@Step @RT(18)S_CheckActiveMoves @F @F @F @F @RT(0) @F
@AcbCont @RT(7)unnamed @F 1
@Acb @RT(19)AGetActiveMovements @F @T @RT(1)P @RT(0) @F @F @T @TL(2)
iActiveMoves := sv_ActiveMovements.iNumberOfActiveMovements;

@F

@AltBranch @RT(3)alt @F 2
@TransSeq @RT(4)tseq @F 1
@Trans @RT(14)TNoMovesActive @F @T @F @F @T @F @TL(2)
iActiveMoves = 0

@RT(7)Trans12 @F

@TransSeq @RT(4)tseq @F 2
@Trans @RT(12)TMovesActive @F @T @F @F @T @F @TL(2)
iActiveMoves > 0

@RT(7)Trans25 @F
@Goto @RT(5)S_End @F @F

@Step @RT(13)S_CheckDemand @F @F @F @F @RT(0) @F
@AcbCont @RT(7)unnamed @F 0

@AltBranch @RT(3)alt @F 2
@TransSeq @RT(4)tseq @F 3
@Trans @RT(14)TLowerHalfAuto @F @T @F @F @T @F @TL(2)
nDemandedMode < nHalfAutomatic

@RT(7)Trans15 @F
@Step @RT(11)S_AllowMode @F @F @F @F @RT(0) @F
@AcbCont @RT(7)unnamed @F 1
@Acb @RT(12)AAllowedMode @F @T @RT(1)P @RT(0) @F @F @T @TL(2)
bAllow := TRUE;

@F

@Trans @RT(7)Trans16 @F @T @F @F @T @F @TL(2)
TRUE

@RT(7)Trans16 @F

@TransSeq @RT(4)tseq @F 5
@Trans @RT(17)TAutoModeDemanded @F @T @F @F @T @F @TL(2)
nDemandedMode > nManual

@RT(7)Trans17 @F
@Step @RT(13)S_CheckAlarms @F @F @F @F @RT(0) @F
@AcbCont @RT(7)unnamed @F 1
@Acb @RT(19)ACheckPendingAlarms @F @F @RT(1)P @RT(0) @F @F @F @F

@AltBranch @RT(3)alt @F 2
@TransSeq @RT(4)tseq @F 1
@Trans @RT(15)TNoActiveAlarms @F @T @F @F @T @F @TL(2)
bPendingAlarmsOk

@RT(7)Trans20 @F

@TransSeq @RT(4)tseq @F 2
@Trans @RT(13)TAcitveAlarms @F @T @F @F @T @F @TL(2)
NOT bPendingAlarmsOk

@RT(7)Trans24 @F
@Goto @RT(5)S_End @F @F

@Step @RT(18)S_CheckAutoAllowed @F @F @F @F @RT(0) @F
@AcbCont @RT(7)unnamed @F 1
@Acb @RT(8)Action15 @F @F @RT(1)P @RT(0) @F @F @F @F

@Trans @RT(7)Trans18 @F @T @F @F @T @F @TL(2)
TRUE

@RT(7)Trans18 @F

@Step @RT(5)S_End @F @F @T @F @RT(0) @F
@AcbCont @RT(7)unnamed @F 1
@Acb @RT(11)ACopyResult @F @T @RT(1)P @RT(0) @F @F @T @TL(2)
bChangeAllowed := bAllow;

@F

@Trans @RT(16)TWaitForNextCall @F @T @T @T @T @T @TL(2)
TRUE

@RT(7)Trans19 @F

@END_SfcData
@SaActions 3
@SaText @RT(6)ACheck 1 @TL(5)
// check if full auto mode is locked
abLockList.aCheck(MoveDir := cModeFullAutomatic,
                  MoveId := cModeFullAutomatic);
bAllow := NOT abLockList.aCheck.bLocked;

@SaText @RT(8)Action15 1 @TL(21)
IF nDemandedMode = nFullAutomatic THEN
    //full auto mode demanded -> check if full auto is locked
    abLockList.aCheck(MoveDir := cModeFullAutomatic,
                        MoveId := cModeFullAutomatic);
    bFullAutoLocked := abLockList.aCheck.bLocked;

    //check if half and full auto is locked
    abLockList.aCheck(MoveDir := cModeAutomatic,
                        MoveId := cModeAutomatic);
    bHalfAutoLocked := abLockList.aCheck.bLocked;

    bAllow := NOT bHalfAutoLocked AND NOT bFullAutoLocked;
ELSIF nDemandedMode = nHalfAutomatic THEN
    //half auto mode demanded
    abLockList.aCheck(MoveDir := cModeAutomatic,
                        MoveId := cModeAutomatic);
    bAllow := NOT abLockList.aCheck.bLocked;
ELSE
    bAllow := TRUE;
END_IF;

@SaText @RT(19)ACheckPendingAlarms 1 @TL(10)
(**************************************** WARNING ********************************************
 *** The KEBA Kemro K2 System including software is not intended for safety control tasks! ***
 ***                       For further information see Comment tab!                        ***
 *********************************************************************************************)

//basically operation mode can not be changed to HA or FA if any alarm of class 1, 2 or 3 is pending
//there is only one exception:
//If the mold safety gate is open it should also be possible to switch to HA and FA
bPendingAlarmsOk := (sv_iPendingAlarms = 0) OR ((sv_iPendingAlarms = 1) AND (sv_MoldSafetyGateState = nOpen));

@SaTrans 0
@SaExits 0
@END_SfcBody

@@@BEG_Comment@@@
@TL(0)

@@@END_Comment@@@
@END_Body

@END_Contents

(* ---- ABOverrideSafetySwitch.pu ---- *)
(*
@h    ! WARNING !
@h    The Kemro K2 system (including software) only meets category B according to EN 954-1,
@h    thus it is not intended for usage in safety-relevant control applications in the field
@h    of personal safety (e.g. emergency stop).
@h    To implement potentially necessary safety-relevant control tasks, always use additional
@h    external safety devices that are intended for the particular purpose, and meet the necessary
@h    functional safety.
@h    For further information see EN 954-1 (EN ISO 13849-1) and/or the K2-x00 user manual, chapter
@h    "CE conformity, directives and standards".

This block handles ejector and core override safety mode.
If OperationMode1.di_CoreEjectorSafetySwitch is linked, the variables system.sv_bOverrideCoreSafety
and system.sv_bOverrideEjectorSafety are set depending on the switch, userlevel and operationmode.
*)

IMPORT_OVER_LISTFILE
 SET_ALARM
, cLevelProcessOperator
, tnOperationMode
, R_TRIG

END_IMPORT

ALGORITHM_BLOCK ABOverrideSafetySwitch #DUMMY_EDIT_BLOCK

SYSTEM_VAR
 sv_bInitDone : BOOL;
 di_CoreEjectorSafetySwitch : BOOL;
 sv_UserLevel : DINT (* actual userlevel *);
 sv_OperationMode : tnOperationMode;
 sv_bOverrideCoreSafety : BOOL (* overrides safety settings for core movements in setup mode *);
 sv_bOverrideEjectorSafety : BOOL (* overrides safety settings for ejector movements in setup mode *);
END_VAR

SYSTEM_OBJECT
 erUserLevelLow : ALARM;
 erSetupModeRequired : ALARM;
 erOverrideSafetyModeOn : ALARM;
 erOverrideSafetyModeOff : ALARM;
 PU_Task_13 : TASK;
END_OBJECT

(*
@h    ! WARNING !
@h    The Kemro K2 system (including software) only meets category B according to EN 954-1,
@h    thus it is not intended for usage in safety-relevant control applications in the field
@h    of personal safety (e.g. emergency stop).
@h    To implement potentially necessary safety-relevant control tasks, always use additional
@h    external safety devices that are intended for the particular purpose, and meet the necessary
@h    functional safety.
@h    For further information see EN 954-1 (EN ISO 13849-1) and/or the K2-x00 user manual, chapter
@h    "CE conformity, directives and standards".

*)

POSTUPDATE_ALGORITHM pOverrideSafettySwitch ON PU_Task_13 WITH di_CoreEjectorSafetySwitch,sv_OperationMode,sv_UserLevel

VAR_TEMP
 bOverrideNew : BOOL;
END_VAR

VAR
 fbRTrigSwitch : R_TRIG;
 bOverrideLast : BOOL;
 bIsDILinked : BOOL;
 bInitDone : BOOL;
END_VAR
#BEGIN_EDIT_BLOCK
(**************************************** WARNING ********************************************
 *** The KEBA Kemro K2 System including software is not intended for safety control tasks! ***
 ***                       For further information see Comment tab!                        ***
 *********************************************************************************************)
IF (NOT bInitDone) THEN
    bIsDILinked := IS_LINKED(di_CoreEjectorSafetySwitch);
    bInitDone := TRUE;
END_IF;

IF (NOT bIsDILinked) THEN
    RETURN;
END_IF;

bOverrideNew := FALSE;

fbRTrigSwitch(CLK := di_CoreEjectorSafetySwitch);

IF (fbRTrigSwitch.Q AND sv_bInitDone) THEN
    IF (sv_UserLevel < cLevelProcessOperator) THEN
        SET_ALARM(Name := erUserLevelLow, Param1 := DINT_TO_INT(cLevelProcessOperator));
    ELSIF (sv_OperationMode <> nSetup)THEN
        SET_ALARM(erSetupModeRequired);
    ELSE
        bOverrideNew := TRUE;
    END_IF;
END_IF;

IF (bOverrideNew AND (NOT bOverrideLast)) THEN
    QUIT_ALARM(erOverrideSafetyModeOff);
    SET_ALARM(erOverrideSafetyModeOn);
END_IF;

IF ((NOT bOverrideNew) AND (bOverrideLast)) THEN
    QUIT_ALARM(erOverrideSafetyModeOn);
    SET_ALARM(erOverrideSafetyModeOff);
END_IF;

sv_bOverrideCoreSafety := bOverrideNew;
sv_bOverrideEjectorSafety := bOverrideNew;
bOverrideLast := bOverrideNew;

;#END_EDIT_BLOCK END_ALGORITHM

END_ALGORITHM_BLOCK

#END_OF_IEC_PART

@Puma @IecEditor 6 131 @Pou 25
@@@BEG_Comment@@@
@h    ! WARNING !
@h    The Kemro K2 system (including software) only meets category B according to EN 954-1,
@h    thus it is not intended for usage in safety-relevant control applications in the field
@h    of personal safety (e.g. emergency stop).
@h    To implement potentially necessary safety-relevant control tasks, always use additional
@h    external safety devices that are intended for the particular purpose, and meet the necessary
@h    functional safety.
@h    For further information see EN 954-1 (EN ISO 13849-1) and/or the K2-x00 user manual, chapter
@h    "CE conformity, directives and standards".

This block handles ejector and core override safety mode.
If OperationMode1.di_CoreEjectorSafetySwitch is linked, the variables system.sv_bOverrideCoreSafety
and system.sv_bOverrideEjectorSafety are set depending on the switch, userlevel and operationmode.
@@@END_Comment@@@

@BEG_Contents

@BEG_Func
@RT(17)FuncTreeContainer
1
@Var @RT(9)SET_ALARM @RT(0) @T @T @DERIVED 0 @F @RT(23)KEBA_STANDARD_PROCEDURE @F
@T
@BEG_Attrib
0 @RT(0) @RT(0)
@END_Attrib
1 1 @F @F @F @F

@END_Func

@BEG_Const
@RT(18)ConstTreeContainer
1
@Var @RT(21)cLevelProcessOperator @RT(0) @T @F @DT @RT(4)DINT @RT(0) @T @T @BASIC 0 @F
@F @F
@T
@BEG_Attrib
0 @RT(1)6 @RT(0)
@END_Attrib
1 1 @F @F @F @F

@END_Const

@BEG_Export

@BEG_Kind
@ALGORITHM_BLOCK @RT(22)ABOverrideSafetySwitch @STRUCTURED_TEXT
@RT(0) @RT(0) @RT(0)
@END_Kind

@BEG_Dcl
@RT(16)DclTreeContainer
11
@Var @RT(12)sv_bInitDone @RT(0) @T @F @DT @RT(4)BOOL @RT(0) @T @T @BASIC 0 @F
@F @F
@T
@BEG_Attrib
3 @RT(0) @RT(0) @RT(0)
@END_Attrib
1 8 @F @F @F @F

@Var @RT(26)di_CoreEjectorSafetySwitch @RT(0) @T @F @DT @RT(4)BOOL @RT(0) @T @T @BASIC 0 @F
@F @F
@T
@BEG_Attrib
3 @RT(0) @RT(0) @RT(0)
@END_Attrib
1 8 @F @F @F @F

@Var @RT(12)sv_UserLevel @RT(0) @T @F @DT @RT(4)DINT @RT(0) @T @T @BASIC 0 @F
@F @F
@T
@BEG_Attrib
3 @RT(0) @RT(16)actual userlevel @RT(0)
@END_Attrib
1 8 @F @F @F @F

@Var @RT(16)sv_OperationMode @RT(0) @T @T @DERIVED 0 @T @T @DT @RT(15)tnOperationMode @RT(0) @T @T @UNKNOWN 0 @F
@F @F
@T
@BEG_Attrib
3 @RT(0) @RT(0) @RT(0)
@END_Attrib
1 8 @F @F @F @F

@Var @RT(22)sv_bOverrideCoreSafety @RT(0) @T @F @DT @RT(4)BOOL @RT(0) @T @T @BASIC 0 @F
@F @F
@T
@BEG_Attrib
3 @RT(0) @RT(58)overrides safety settings for core movements in setup mode @RT(0)
@END_Attrib
1 8 @F @F @F @F

@Var @RT(25)sv_bOverrideEjectorSafety @RT(0) @T @F @DT @RT(4)BOOL @RT(0) @T @T @BASIC 0 @F
@F @F
@T
@BEG_Attrib
3 @RT(0) @RT(61)overrides safety settings for ejector movements in setup mode @RT(0)
@END_Attrib
1 8 @F @F @F @F

@Var @RT(14)erUserLevelLow @RT(0) @T @F @DT @RT(5)ALARM @RT(0) @T @T @BASIC 0 @F
@F @F
@T
@BEG_Attrib
3 @RT(0) @RT(0) @RT(0)
@END_Attrib
1 7 @F @F @F @F

@Var @RT(19)erSetupModeRequired @RT(0) @T @F @DT @RT(5)ALARM @RT(0) @T @T @BASIC 0 @F
@F @F
@T
@BEG_Attrib
3 @RT(0) @RT(0) @RT(0)
@END_Attrib
1 7 @F @F @F @F

@Var @RT(22)erOverrideSafetyModeOn @RT(0) @T @F @DT @RT(5)ALARM @RT(0) @T @T @BASIC 0 @F
@F @F
@T
@BEG_Attrib
3 @RT(0) @RT(0) @RT(0)
@END_Attrib
1 7 @F @F @F @F

@Var @RT(23)erOverrideSafetyModeOff @RT(0) @T @F @DT @RT(5)ALARM @RT(0) @T @T @BASIC 0 @F
@F @F
@T
@BEG_Attrib
3 @RT(0) @RT(0) @RT(0)
@END_Attrib
1 7 @F @F @F @F

@Var @RT(10)PU_Task_13 @RT(0) @T @F @DT @RT(4)TASK @RT(0) @T @T @BASIC 0 @F
@F @F
@T
@BEG_Attrib
3 @RT(0) @RT(0) @RT(0)
@END_Attrib
1 7 @F @F @F @F

@END_Dcl

@END_Export

@BEG_Body

1

@BEG_Export

@BEG_Algo
@POSTUPDATE_ALGORITHM @RT(22)pOverrideSafettySwitch @STRUCTURED_TEXT
@RT(0) @RT(56)di_CoreEjectorSafetySwitch,sv_OperationMode,sv_UserLevel @RT(10)PU_Task_13 @F @F
@END_Algo

@BEG_Dcl
@RT(16)DclTreeContainer
5
@Var @RT(12)bOverrideNew @RT(0) @T @F @DT @RT(4)BOOL @RT(0) @T @T @BASIC 0 @F
@F @F
@T
@BEG_Attrib
3 @RT(0) @RT(0) @RT(0)
@END_Attrib
1 4 @F @F @F @F

@Var @RT(13)fbRTrigSwitch @RT(0) @T @T @DERIVED 0 @F @RT(6)R_TRIG @F
@T
@BEG_Attrib
3 @RT(0) @RT(0) @RT(0)
@END_Attrib
1 0 @F @F @F @F

@Var @RT(13)bOverrideLast @RT(0) @T @F @DT @RT(4)BOOL @RT(0) @T @T @BASIC 0 @F
@F @F
@T
@BEG_Attrib
3 @RT(0) @RT(0) @RT(0)
@END_Attrib
1 0 @F @F @F @F

@Var @RT(11)bIsDILinked @RT(0) @T @F @DT @RT(4)BOOL @RT(0) @T @T @BASIC 0 @F
@F @F
@T
@BEG_Attrib
3 @RT(0) @RT(0) @RT(0)
@END_Attrib
1 0 @F @F @F @F

@Var @RT(9)bInitDone @RT(0) @T @F @DT @RT(4)BOOL @RT(0) @T @T @BASIC 0 @F
@F @F
@T
@BEG_Attrib
3 @RT(0) @RT(0) @RT(0)
@END_Attrib
1 0 @F @F @F @F

@END_Dcl

@END_Export

@BEG_Body
@TL(42)
(**************************************** WARNING ********************************************
 *** The KEBA Kemro K2 System including software is not intended for safety control tasks! ***
 ***                       For further information see Comment tab!                        ***
 *********************************************************************************************)
IF (NOT bInitDone) THEN
    bIsDILinked := IS_LINKED(di_CoreEjectorSafetySwitch);
    bInitDone := TRUE;
END_IF;

IF (NOT bIsDILinked) THEN
    RETURN;
END_IF;

bOverrideNew := FALSE;

fbRTrigSwitch(CLK := di_CoreEjectorSafetySwitch);

IF (fbRTrigSwitch.Q AND sv_bInitDone) THEN
    IF (sv_UserLevel < cLevelProcessOperator) THEN
        SET_ALARM(Name := erUserLevelLow, Param1 := DINT_TO_INT(cLevelProcessOperator));
    ELSIF (sv_OperationMode <> nSetup)THEN
        SET_ALARM(erSetupModeRequired);
    ELSE
        bOverrideNew := TRUE;
    END_IF;
END_IF;

IF (bOverrideNew AND (NOT bOverrideLast)) THEN
    QUIT_ALARM(erOverrideSafetyModeOff);
    SET_ALARM(erOverrideSafetyModeOn);
END_IF;

IF ((NOT bOverrideNew) AND (bOverrideLast)) THEN
    QUIT_ALARM(erOverrideSafetyModeOn);
    SET_ALARM(erOverrideSafetyModeOff);
END_IF;

sv_bOverrideCoreSafety := bOverrideNew;
sv_bOverrideEjectorSafety := bOverrideNew;
bOverrideLast := bOverrideNew;

@END_Body

@@@BEG_Comment@@@
@TL(10)
@h    ! WARNING !
@h    The Kemro K2 system (including software) only meets category B according to EN 954-1,
@h    thus it is not intended for usage in safety-relevant control applications in the field
@h    of personal safety (e.g. emergency stop).
@h    To implement potentially necessary safety-relevant control tasks, always use additional
@h    external safety devices that are intended for the particular purpose, and meet the necessary
@h    functional safety.
@h    For further information see EN 954-1 (EN ISO 13849-1) and/or the K2-x00 user manual, chapter
@h    "CE conformity, directives and standards".

@@@END_Comment@@@
@END_Body

@END_Contents
